LIN {X 0,Y 370.428,Z 641.717,A -85,B 0,C 180,E1 -12894.345,E2 -12894.345} C_VEL
LIN {X 0,Y 371.468,Z 578.131,A -85,B 0,C 180,E1 -12895.586,E2 -12895.586} C_VEL
LIN {X 0,Y 367.34,Z 559.666,A -85,B 0,C 180,E1 -12896.25,E2 -12896.25} C_VEL
LIN {X 0,Y 364.561,Z 552.172,A -85,B 0,C 180,E1 -12896.629,E2 -12896.629} C_VEL
LIN {X 0,Y 362.723,Z 543.261,A -85,B 0,C 180,E1 -12899.318,E2 -12899.318} C_VEL
LIN {X 0,Y 361.889,Z 539.398,A -85,B 0,C 180,E1 -12900.555,E2 -12900.555} C_VEL
LIN {X 0,Y 361.854,Z 539.415,A -85,B 0,C 180,E1 -12904.279,E2 -12904.279} C_VEL
LIN {X 0,Y 361.865,Z 539.408,A -85,B 0,C 180,E1 -12907.222,E2 -12907.222} C_VEL
LIN {X 0,Y 361.904,Z 539.408,A -85,B 0,C 180,E1 -12910.767,E2 -12910.767} C_VEL
LIN {X 0,Y 361.909,Z 539.405,A -85,B 0,C 180,E1 -12914.353,E2 -12914.353} C_VEL
LIN {X 0,Y 361.854,Z 539.407,A -85,B 0,C 180,E1 -12917.563,E2 -12917.563} C_VEL
LIN {X 0,Y 361.87,Z 539.41,A -85,B 0,C 180,E1 -12920.972,E2 -12920.972} C_VEL
LIN {X 0,Y 361.87,Z 539.412,A -85,B 0,C 180,E1 -12924.654,E2 -12924.654} C_VEL
LIN {X 0,Y 361.833,Z 539.415,A -85,B 0,C 180,E1 -12928.37,E2 -12928.37} C_VEL
LIN {X 0,Y 361.897,Z 539.407,A -85,B 0,C 180,E1 -12930.955,E2 -12930.955} C_VEL
LIN {X 0,Y 361.949,Z 539.391,A -85,B 0,C 180,E1 -12933.474,E2 -12933.474} C_VEL
LIN {X 0,Y 361.883,Z 539.4,A -85,B 0,C 180,E1 -12937.144,E2 -12937.144} C_VEL
LIN {X 0,Y 361.899,Z 539.405,A -85,B 0,C 180,E1 -12940.723,E2 -12940.723} C_VEL
LIN {X 0,Y 361.925,Z 539.4,A -85,B 0,C 180,E1 -12943.065,E2 -12943.065} C_VEL
LIN {X 0,Y 361.991,Z 539.389,A -85,B 0,C 180,E1 -12946.527,E2 -12946.527} C_VEL
LIN {X 0,Y 362.024,Z 539.388,A -85,B 0,C 180,E1 -12949.938,E2 -12949.938} C_VEL
LIN {X 0,Y 362.155,Z 539.368,A -85,B 0,C 180,E1 -12953.313,E2 -12953.313} C_VEL
LIN {X 0,Y 362.275,Z 539.348,A -85,B 0,C 180,E1 -12957.776,E2 -12957.776} C_VEL
LIN {X 0,Y 362.421,Z 539.338,A -85,B 0,C 180,E1 -12960,E2 -12960} C_VEL
LIN {X 0,Y 362.274,Z 539.357,A -85,B 0,C 180,E1 -12962.223,E2 -12962.223} C_VEL
LIN {X 0,Y 362.154,Z 539.373,A -85,B 0,C 180,E1 -12966.686,E2 -12966.686} C_VEL
LIN {X 0,Y 362.023,Z 539.385,A -85,B 0,C 180,E1 -12970.062,E2 -12970.062} C_VEL
LIN {X 0,Y 361.99,Z 539.384,A -85,B 0,C 180,E1 -12973.899,E2 -12973.899} C_VEL
LIN {X 0,Y 361.96,Z 539.393,A -85,B 0,C 180,E1 -12977.939,E2 -12977.939} C_VEL
LIN {X 0,Y 361.854,Z 539.408,A -85,B 0,C 180,E1 -12981.655,E2 -12981.655} C_VEL
LIN {X 0,Y 361.92,Z 539.4,A -85,B 0,C 180,E1 -12985.291,E2 -12985.291} C_VEL
LIN {X 0,Y 361.916,Z 539.395,A -85,B 0,C 180,E1 -12987.778,E2 -12987.778} C_VEL
LIN {X 0,Y 361.841,Z 539.41,A -85,B 0,C 180,E1 -12991.286,E2 -12991.286} C_VEL
LIN {X 0,Y 361.849,Z 539.412,A -85,B 0,C 180,E1 -12994.281,E2 -12994.281} C_VEL
LIN {X 0,Y 361.86,Z 539.408,A -85,B 0,C 180,E1 -12997.224,E2 -12997.224} C_VEL
LIN {X 0,Y 361.868,Z 539.411,A -85,B 0,C 180,E1 -13000.763,E2 -13000.763} C_VEL
LIN {X 0,Y 361.861,Z 539.412,A -85,B 0,C 180,E1 -13004.362,E2 -13004.362} C_VEL
LIN {X 0,Y 361.833,Z 539.413,A -85,B 0,C 180,E1 -13007.569,E2 -13007.569} C_VEL
LIN {X 0,Y 361.868,Z 539.411,A -85,B 0,C 180,E1 -13010.974,E2 -13010.974} C_VEL
LIN {X 0,Y 361.872,Z 539.408,A -85,B 0,C 180,E1 -13014.656,E2 -13014.656} C_VEL
LIN {X 0,Y 361.836,Z 539.416,A -85,B 0,C 180,E1 -13018.371,E2 -13018.371} C_VEL
LIN {X 0,Y 361.912,Z 539.551,A -85,B 0,C 180,E1 -13019.371,E2 -13019.371} C_VEL
LIN {X 0,Y 364.641,Z 551.604,A -85,B 0,C 180,E1 -13022.698,E2 -13022.698} C_VEL
LIN {X 0,Y 366.223,Z 560.485,A -85,B 0,C 180,E1 -13025.028,E2 -13025.028} C_VEL
LIN {X 0,Y 365.183,Z 571.057,A -85,B 0,C 180,E1 -13027.484,E2 -13027.484} C_VEL
LIN {X 0,Y 370.275,Z 598.191,A -85,B 0,C 180,E1 -13028.394,E2 -13028.394} C_VEL
LIN {X 0,Y 371.148,Z 604.978,A -85,B 0,C 180,E1 -13028.591,E2 -13028.591} C_VEL
LIN {X 0,Y 369.787,Z 679.549,A -85,B 0,C 180,E1 -13030.068,E2 -13030.068} C_VEL
LIN {X 0,Y 369.085,Z 693.347,A -85,B 0,C 180,E1 -13030.572,E2 -13030.572} C_VEL
LIN {X 0,Y 368.192,Z 705.186,A -85,B 0,C 180,E1 -13031.21,E2 -13031.21} C_VEL
LIN {X 0,Y 367.163,Z 716.398,A -85,B 0,C 180,E1 -13032.022,E2 -13032.022} C_VEL
LIN {X 0,Y 365.9,Z 728.011,A -85,B 0,C 180,E1 -13033.112,E2 -13033.112} C_VEL
LIN {X 0,Y 364.719,Z 738.465,A -85,B 0,C 180,E1 -13034.35,E2 -13034.35} C_VEL
LIN {X 0,Y 363.708,Z 747.897,A -85,B 0,C 180,E1 -13035.738,E2 -13035.738} C_VEL
LIN {X 0,Y 362.56,Z 756.994,A -85,B 0,C 180,E1 -13037.404,E2 -13037.404} C_VEL
LIN {X 0,Y 361.706,Z 764.336,A -85,B 0,C 180,E1 -13039.08,E2 -13039.08} C_VEL
LIN {X 0,Y 361.013,Z 771.091,A -85,B 0,C 180,E1 -13041.041,E2 -13041.041} C_VEL
LIN {X 0,Y 360.601,Z 775.559,A -85,B 0,C 180,E1 -13042.722,E2 -13042.722} C_VEL
LIN {X 0,Y 360.383,Z 778.956,A -85,B 0,C 180,E1 -13044.404,E2 -13044.404} C_VEL
LIN {X 0,Y 360.368,Z 780.651,A -85,B 0,C 180,E1 -13045.526,E2 -13045.526} C_VEL
LIN {X 0,Y 360.3,Z 781.942,A -85,B 0,C 180,E1 -13046.645,E2 -13046.645} C_VEL
LIN {X 0,Y 360.263,Z 782.842,A -85,B 0,C 180,E1 -13047.764,E2 -13047.764} C_VEL
LIN {X 0,Y 360.316,Z 783.319,A -85,B 0,C 180,E1 -13048.882,E2 -13048.882} C_VEL
LIN {X 0,Y 360.359,Z 783.388,A -85,B 0,C 180,E1 -13050,E2 -13050} C_VEL
LIN {X 0,Y 360.317,Z 783.068,A -85,B 0,C 180,E1 -13051.118,E2 -13051.118} C_VEL
LIN {X 0,Y 360.267,Z 782.362,A -85,B 0,C 180,E1 -13052.236,E2 -13052.236} C_VEL
LIN {X 0,Y 360.302,Z 781.236,A -85,B 0,C 180,E1 -13053.355,E2 -13053.355} C_VEL
LIN {X 0,Y 360.368,Z 779.672,A -85,B 0,C 180,E1 -13054.474,E2 -13054.474} C_VEL
LIN {X 0,Y 360.38,Z 776.953,A -85,B 0,C 180,E1 -13055.964,E2 -13055.964} C_VEL
LIN {X 0,Y 360.672,Z 772.311,A -85,B 0,C 180,E1 -13057.839,E2 -13057.839} C_VEL
LIN {X 0,Y 361.163,Z 765.895,A -85,B 0,C 180,E1 -13059.803,E2 -13059.803} C_VEL
LIN {X 0,Y 361.776,Z 758.895,A -85,B 0,C 180,E1 -13061.485,E2 -13061.485} C_VEL
LIN {X 0,Y 362.736,Z 750.12,A -85,B 0,C 180,E1 -13063.159,E2 -13063.159} C_VEL
LIN {X 0,Y 363.645,Z 741.125,A -85,B 0,C 180,E1 -13064.551,E2 -13064.551} C_VEL
LIN {X 0,Y 364.512,Z 731.227,A -85,B 0,C 180,E1 -13065.803,E2 -13065.803} C_VEL
LIN {X 0,Y 365.496,Z 720.293,A -85,B 0,C 180,E1 -13066.907,E2 -13066.907} C_VEL
LIN {X 0,Y 366.567,Z 708.023,A -85,B 0,C 180,E1 -13067.864,E2 -13067.864} C_VEL
LIN {X 0,Y 367.327,Z 696.44,A -85,B 0,C 180,E1 -13068.547,E2 -13068.547} C_VEL
LIN {X 0,Y 367.994,Z 684.292,A -85,B 0,C 180,E1 -13069.053,E2 -13069.053} C_VEL
LIN {X 0,Y 368.341,Z 670.698,A -85,B 0,C 180,E1 -13069.397,E2 -13069.397} C_VEL
LIN {X 0,Y 369.31,Z 603.202,A -85,B 0,C 180,E1 -13070.703,E2 -13070.703} C_VEL
LIN {X 0,Y 364.289,Z 570.9,A -85,B 0,C 180,E1 -13071.65,E2 -13071.65} C_VEL
LIN {X 0,Y 365.458,Z 558.977,A -85,B 0,C 180,E1 -13074.422,E2 -13074.422} C_VEL
LIN {X 0,Y 364.826,Z 553.825,A -85,B 0,C 180,E1 -13075.697,E2 -13075.697} C_VEL
LIN {X 0,Y 362.245,Z 541.043,A -85,B 0,C 180,E1 -13079.014,E2 -13079.014} C_VEL
LIN {X 0,Y 361.912,Z 539.406,A -85,B 0,C 180,E1 -13079.505,E2 -13079.505} C_VEL
LIN {X 0,Y 361.857,Z 539.412,A -85,B 0,C 180,E1 -13083.369,E2 -13083.369} C_VEL
LIN {X 0,Y 361.87,Z 539.407,A -85,B 0,C 180,E1 -13087.017,E2 -13087.017} C_VEL
LIN {X 0,Y 361.853,Z 539.41,A -85,B 0,C 180,E1 -13089.86,E2 -13089.86} C_VEL
LIN {X 0,Y 361.833,Z 539.411,A -85,B 0,C 180,E1 -13092.828,E2 -13092.828} C_VEL
LIN {X 0,Y 361.853,Z 539.409,A -85,B 0,C 180,E1 -13095.939,E2 -13095.939} C_VEL
LIN {X 0,Y 361.868,Z 539.409,A -85,B 0,C 180,E1 -13099.237,E2 -13099.237} C_VEL
LIN {X 0,Y 361.864,Z 539.408,A -85,B 0,C 180,E1 -13102.982,E2 -13102.982} C_VEL
LIN {X 0,Y 361.853,Z 539.407,A -85,B 0,C 180,E1 -13106.63,E2 -13106.63} C_VEL
LIN {X 0,Y 361.87,Z 539.409,A -85,B 0,C 180,E1 -13109.672,E2 -13109.672} C_VEL
LIN {X 0,Y 361.948,Z 539.402,A -85,B 0,C 180,E1 -13113.475,E2 -13113.475} C_VEL
LIN {X 0,Y 361.875,Z 539.408,A -85,B 0,C 180,E1 -13117.144,E2 -13117.144} C_VEL
LIN {X 0,Y 361.913,Z 539.4,A -85,B 0,C 180,E1 -13120.724,E2 -13120.724} C_VEL
LIN {X 0,Y 361.938,Z 539.397,A -85,B 0,C 180,E1 -13124.226,E2 -13124.226} C_VEL
LIN {X 0,Y 361.991,Z 539.39,A -85,B 0,C 180,E1 -13126.528,E2 -13126.528} C_VEL
LIN {X 0,Y 362.023,Z 539.388,A -85,B 0,C 180,E1 -13129.938,E2 -13129.938} C_VEL
LIN {X 0,Y 362.156,Z 539.375,A -85,B 0,C 180,E1 -13133.314,E2 -13133.314} C_VEL
LIN {X 0,Y 362.275,Z 539.358,A -85,B 0,C 180,E1 -13137.777,E2 -13137.777} C_VEL
LIN {X 0,Y 362.419,Z 539.338,A -85,B 0,C 180,E1 -13140,E2 -13140} C_VEL
LIN {X 0,Y 362.275,Z 539.355,A -85,B 0,C 180,E1 -13142.224,E2 -13142.224} C_VEL
LIN {X 0,Y 362.156,Z 539.37,A -85,B 0,C 180,E1 -13146.687,E2 -13146.687} C_VEL
LIN {X 0,Y 362.024,Z 539.387,A -85,B 0,C 180,E1 -13150.062,E2 -13150.062} C_VEL
LIN {X 0,Y 361.99,Z 539.392,A -85,B 0,C 180,E1 -13153.899,E2 -13153.899} C_VEL
LIN {X 0,Y 361.96,Z 539.395,A -85,B 0,C 180,E1 -13157.939,E2 -13157.939} C_VEL
LIN {X 0,Y 361.887,Z 539.407,A -85,B 0,C 180,E1 -13161.654,E2 -13161.654} C_VEL
LIN {X 0,Y 361.922,Z 539.404,A -85,B 0,C 180,E1 -13165.291,E2 -13165.291} C_VEL
LIN {X 0,Y 361.917,Z 539.402,A -85,B 0,C 180,E1 -13167.779,E2 -13167.779} C_VEL
LIN {X 0,Y 361.842,Z 539.414,A -85,B 0,C 180,E1 -13171.286,E2 -13171.286} C_VEL
LIN {X 0,Y 361.85,Z 539.408,A -85,B 0,C 180,E1 -13174.281,E2 -13174.281} C_VEL
LIN {X 0,Y 361.867,Z 539.41,A -85,B 0,C 180,E1 -13177.225,E2 -13177.225} C_VEL
LIN {X 0,Y 361.833,Z 539.411,A -85,B 0,C 180,E1 -13180.757,E2 -13180.757} C_VEL
LIN {X 0,Y 361.844,Z 539.408,A -85,B 0,C 180,E1 -13184.365,E2 -13184.365} C_VEL
LIN {X 0,Y 361.882,Z 539.409,A -85,B 0,C 180,E1 -13187.561,E2 -13187.561} C_VEL
LIN {X 0,Y 361.874,Z 539.407,A -85,B 0,C 180,E1 -13190.973,E2 -13190.973} C_VEL
LIN {X 0,Y 361.874,Z 539.405,A -85,B 0,C 180,E1 -13194.656,E2 -13194.656} C_VEL
LIN {X 0,Y 361.837,Z 539.409,A -85,B 0,C 180,E1 -13198.371,E2 -13198.371} C_VEL
LIN {X 0,Y 361.901,Z 539.403,A -85,B 0,C 180,E1 -13200.956,E2 -13200.956} C_VEL
LIN {X 0,Y 361.956,Z 539.4,A -85,B 0,C 180,E1 -13203.476,E2 -13203.476} C_VEL
LIN {X 0,Y 361.892,Z 539.406,A -85,B 0,C 180,E1 -13207.145,E2 -13207.145} C_VEL
LIN {X 0,Y 361.903,Z 539.507,A -85,B 0,C 180,E1 -13208.772,E2 -13208.772} C_VEL
LIN {X 0,Y 363.757,Z 548.685,A -85,B 0,C 180,E1 -13211.465,E2 -13211.465} C_VEL
LIN {X 0,Y 364.348,Z 552.074,A -85,B 0,C 180,E1 -13212.431,E2 -13212.431} C_VEL
LIN {X 0,Y 366.507,Z 560.951,A -85,B 0,C 180,E1 -13212.742,E2 -13212.742} C_VEL
LIN {X 0,Y 369.698,Z 577.539,A -85,B 0,C 180,E1 -13213.256,E2 -13213.256} C_VEL
LIN {X 0,Y 368.433,Z 659.251,A -85,B 0,C 180,E1 -13214.865,E2 -13214.865} C_VEL
LIN {X 0,Y 367.932,Z 671.574,A -85,B 0,C 180,E1 -13215.304,E2 -13215.304} C_VEL
LIN {X 0,Y 367.179,Z 684.929,A -85,B 0,C 180,E1 -13216.016,E2 -13216.016} C_VEL
LIN {X 0,Y 366.354,Z 696.143,A -85,B 0,C 180,E1 -13216.832,E2 -13216.832} C_VEL
LIN {X 0,Y 365.456,Z 707.705,A -85,B 0,C 180,E1 -13217.929,E2 -13217.929} C_VEL
LIN {X 0,Y 364.341,Z 718.119,A -85,B 0,C 180,E1 -13219.16,E2 -13219.16} C_VEL
LIN {X 0,Y 363.471,Z 726.919,A -85,B 0,C 180,E1 -13220.447,E2 -13220.447} C_VEL
LIN {X 0,Y 362.708,Z 735.175,A -85,B 0,C 180,E1 -13221.925,E2 -13221.925} C_VEL
LIN {X 0,Y 361.952,Z 742.691,A -85,B 0,C 180,E1 -13223.59,E2 -13223.59} C_VEL
LIN {X 0,Y 361.489,Z 747.841,A -85,B 0,C 180,E1 -13224.981,E2 -13224.981} C_VEL
LIN {X 0,Y 360.912,Z 752.837,A -85,B 0,C 180,E1 -13226.651,E2 -13226.651} C_VEL
LIN {X 0,Y 360.63,Z 756.711,A -85,B 0,C 180,E1 -13228.325,E2 -13228.325} C_VEL
LIN {X 0,Y 360.435,Z 759.571,A -85,B 0,C 180,E1 -13230,E2 -13230} C_VEL
LIN {X 0,Y 360.372,Z 760.923,A -85,B 0,C 180,E1 -13231.117,E2 -13231.117} C_VEL
LIN {X 0,Y 360.307,Z 762.469,A -85,B 0,C 180,E1 -13233.355,E2 -13233.355} C_VEL
LIN {X 0,Y 360.337,Z 762.65,A -85,B 0,C 180,E1 -13234.474,E2 -13234.474} C_VEL
LIN {X 0,Y 360.387,Z 761.791,A -85,B 0,C 180,E1 -13236.719,E2 -13236.719} C_VEL
LIN {X 0,Y 360.458,Z 760.786,A -85,B 0,C 180,E1 -13237.844,E2 -13237.844} C_VEL
LIN {X 0,Y 360.563,Z 759.362,A -85,B 0,C 180,E1 -13238.971,E2 -13238.971} C_VEL
LIN {X 0,Y 360.819,Z 756.409,A -85,B 0,C 180,E1 -13240.663,E2 -13240.663} C_VEL
LIN {X 0,Y 361.301,Z 752.402,A -85,B 0,C 180,E1 -13242.355,E2 -13242.355} C_VEL
LIN {X 0,Y 361.886,Z 747.191,A -85,B 0,C 180,E1 -13244.057,E2 -13244.057} C_VEL
LIN {X 0,Y 362.686,Z 740.685,A -85,B 0,C 180,E1 -13245.74,E2 -13245.74} C_VEL
LIN {X 0,Y 363.732,Z 732.542,A -85,B 0,C 180,E1 -13247.427,E2 -13247.427} C_VEL
LIN {X 0,Y 364.811,Z 724.201,A -85,B 0,C 180,E1 -13248.825,E2 -13248.825} C_VEL
LIN {X 0,Y 365.93,Z 713.912,A -85,B 0,C 180,E1 -13250.224,E2 -13250.224} C_VEL
LIN {X 0,Y 367.195,Z 702.254,A -85,B 0,C 180,E1 -13251.471,E2 -13251.471} C_VEL
LIN {X 0,Y 368.295,Z 690.699,A -85,B 0,C 180,E1 -13252.435,E2 -13252.435} C_VEL
LIN {X 0,Y 369.137,Z 678.654,A -85,B 0,C 180,E1 -13253.195,E2 -13253.195} C_VEL
LIN {X 0,Y 369.331,Z 674.63,A -85,B 0,C 180,E1 -13253.406,E2 -13253.406} C_VEL
LIN {X 0,Y 369.243,Z 668.987,A -85,B 0,C 180,E1 -13253.678,E2 -13253.678} C_VEL
LIN {X 0,Y 367.049,Z 659.817,A -85,B 0,C 180,E1 -13254.149,E2 -13254.149} C_VEL
LIN {X 0,Y 364.45,Z 650.556,A -85,B 0,C 180,E1 -13254.544,E2 -13254.544} C_VEL
LIN {X 0,Y 363.836,Z 644.759,A -85,B 0,C 180,E1 -13254.703,E2 -13254.703} C_VEL
LIN {X 0,Y 364.96,Z 579.185,A -85,B 0,C 180,E1 -13256.005,E2 -13256.005} C_VEL
LIN {X 0,Y 361.216,Z 562.272,A -85,B 0,C 180,E1 -13256.628,E2 -13256.628} C_VEL
LIN {X 0,Y 357.409,Z 552.439,A -85,B 0,C 180,E1 -13257.132,E2 -13257.132} C_VEL
LIN {X 0,Y 355.718,Z 544.387,A -85,B 0,C 180,E1 -13259.62,E2 -13259.62} C_VEL
LIN {X 0,Y 354.829,Z 540.277,A -85,B 0,C 180,E1 -13260.995,E2 -13260.995} C_VEL
LIN {X 0,Y 354.812,Z 540.287,A -85,B 0,C 180,E1 -13265.058,E2 -13265.058} C_VEL
LIN {X 0,Y 354.807,Z 540.285,A -85,B 0,C 180,E1 -13267.882,E2 -13267.882} C_VEL
LIN {X 0,Y 354.837,Z 540.284,A -85,B 0,C 180,E1 -13271.18,E2 -13271.18} C_VEL
LIN {X 0,Y 354.861,Z 540.284,A -85,B 0,C 180,E1 -13274.522,E2 -13274.522} C_VEL
LIN {X 0,Y 354.811,Z 540.284,A -85,B 0,C 180,E1 -13277.665,E2 -13277.665} C_VEL
LIN {X 0,Y 354.834,Z 540.283,A -85,B 0,C 180,E1 -13280.668,E2 -13280.668} C_VEL
LIN {X 0,Y 354.818,Z 540.287,A -85,B 0,C 180,E1 -13284.3,E2 -13284.3} C_VEL
LIN {X 0,Y 354.782,Z 540.29,A -85,B 0,C 180,E1 -13287.666,E2 -13287.666} C_VEL
LIN {X 0,Y 354.864,Z 540.28,A -85,B 0,C 180,E1 -13290.62,E2 -13290.62} C_VEL
LIN {X 0,Y 354.893,Z 540.272,A -85,B 0,C 180,E1 -13294.172,E2 -13294.172} C_VEL
LIN {X 0,Y 354.828,Z 540.277,A -85,B 0,C 180,E1 -13297.893,E2 -13297.893} C_VEL
LIN {X 0,Y 354.915,Z 540.269,A -85,B 0,C 180,E1 -13301.891,E2 -13301.891} C_VEL
LIN {X 0,Y 354.935,Z 540.27,A -85,B 0,C 180,E1 -13305.981,E2 -13305.981} C_VEL
LIN {X 0,Y 354.97,Z 540.266,A -85,B 0,C 180,E1 -13309.735,E2 -13309.735} C_VEL
LIN {X 0,Y 355.118,Z 540.246,A -85,B 0,C 180,E1 -13313.18,E2 -13313.18} C_VEL
LIN {X 0,Y 355.238,Z 540.224,A -85,B 0,C 180,E1 -13317.732,E2 -13317.732} C_VEL
LIN {X 0,Y 355.391,Z 540.213,A -85,B 0,C 180,E1 -13320,E2 -13320} C_VEL
LIN {X 0,Y 355.238,Z 540.232,A -85,B 0,C 180,E1 -13322.268,E2 -13322.268} C_VEL
LIN {X 0,Y 355.118,Z 540.248,A -85,B 0,C 180,E1 -13326.819,E2 -13326.819} C_VEL
LIN {X 0,Y 354.97,Z 540.266,A -85,B 0,C 180,E1 -13330.264,E2 -13330.264} C_VEL
LIN {X 0,Y 354.935,Z 540.263,A -85,B 0,C 180,E1 -13334.019,E2 -13334.019} C_VEL
LIN {X 0,Y 354.916,Z 540.271,A -85,B 0,C 180,E1 -13338.109,E2 -13338.109} C_VEL
LIN {X 0,Y 354.809,Z 540.287,A -85,B 0,C 180,E1 -13342.108,E2 -13342.108} C_VEL
LIN {X 0,Y 354.892,Z 540.276,A -85,B 0,C 180,E1 -13345.828,E2 -13345.828} C_VEL
LIN {X 0,Y 354.848,Z 540.281,A -85,B 0,C 180,E1 -13349.679,E2 -13349.679} C_VEL
LIN {X 0,Y 354.801,Z 540.287,A -85,B 0,C 180,E1 -13353.703,E2 -13353.703} C_VEL
LIN {X 0,Y 354.794,Z 540.292,A -85,B 0,C 180,E1 -13356.46,E2 -13356.46} C_VEL
LIN {X 0,Y 354.819,Z 540.285,A -85,B 0,C 180,E1 -13359.424,E2 -13359.424} C_VEL
LIN {X 0,Y 354.801,Z 540.292,A -85,B 0,C 180,E1 -13362.871,E2 -13362.871} C_VEL
LIN {X 0,Y 354.766,Z 540.294,A -85,B 0,C 180,E1 -13366.105,E2 -13366.105} C_VEL
LIN {X 0,Y 354.786,Z 540.291,A -85,B 0,C 180,E1 -13369.18,E2 -13369.18} C_VEL
LIN {X 0,Y 354.806,Z 540.287,A -85,B 0,C 180,E1 -13372.403,E2 -13372.403} C_VEL
LIN {X 0,Y 354.81,Z 540.289,A -85,B 0,C 180,E1 -13374.942,E2 -13374.942} C_VEL
LIN {X 0,Y 354.832,Z 540.386,A -85,B 0,C 180,E1 -13378.923,E2 -13378.923} C_VEL
LIN {X 0,Y 357.509,Z 551.94,A -85,B 0,C 180,E1 -13382.205,E2 -13382.205} C_VEL
LIN {X 0,Y 359.308,Z 561.667,A -85,B 0,C 180,E1 -13384.823,E2 -13384.823} C_VEL
LIN {X 0,Y 358.399,Z 570.588,A -85,B 0,C 180,E1 -13386.987,E2 -13386.987} C_VEL
LIN {X 0,Y 363.845,Z 599.803,A -85,B 0,C 180,E1 -13387.997,E2 -13387.997} C_VEL
LIN {X 0,Y 364.603,Z 606.653,A -85,B 0,C 180,E1 -13388.193,E2 -13388.193} C_VEL
LIN {X 0,Y 363.197,Z 679.224,A -85,B 0,C 180,E1 -13389.654,E2 -13389.654} C_VEL
LIN {X 0,Y 362.483,Z 693.061,A -85,B 0,C 180,E1 -13390.166,E2 -13390.166} C_VEL
LIN {X 0,Y 361.485,Z 705.467,A -85,B 0,C 180,E1 -13390.848,E2 -13390.848} C_VEL
LIN {X 0,Y 360.263,Z 718.124,A -85,B 0,C 180,E1 -13391.813,E2 -13391.813} C_VEL
LIN {X 0,Y 358.959,Z 729.382,A -85,B 0,C 180,E1 -13392.922,E2 -13392.922} C_VEL
LIN {X 0,Y 357.738,Z 739.73,A -85,B 0,C 180,E1 -13394.211,E2 -13394.211} C_VEL
LIN {X 0,Y 356.614,Z 749.505,A -85,B 0,C 180,E1 -13395.739,E2 -13395.739} C_VEL
LIN {X 0,Y 355.429,Z 758.294,A -85,B 0,C 180,E1 -13397.438,E2 -13397.438} C_VEL
LIN {X 0,Y 354.59,Z 765.335,A -85,B 0,C 180,E1 -13399.147,E2 -13399.147} C_VEL
LIN {X 0,Y 353.96,Z 770.973,A -85,B 0,C 180,E1 -13400.86,E2 -13400.86} C_VEL
LIN {X 0,Y 353.525,Z 775.421,A -85,B 0,C 180,E1 -13402.576,E2 -13402.576} C_VEL
LIN {X 0,Y 353.281,Z 778.799,A -85,B 0,C 180,E1 -13404.292,E2 -13404.292} C_VEL
LIN {X 0,Y 353.28,Z 780.485,A -85,B 0,C 180,E1 -13405.436,E2 -13405.436} C_VEL
LIN {X 0,Y 353.222,Z 781.768,A -85,B 0,C 180,E1 -13406.578,E2 -13406.578} C_VEL
LIN {X 0,Y 353.172,Z 782.658,A -85,B 0,C 180,E1 -13407.719,E2 -13407.719} C_VEL
LIN {X 0,Y 353.216,Z 783.119,A -85,B 0,C 180,E1 -13408.86,E2 -13408.86} C_VEL
LIN {X 0,Y 353.262,Z 783.179,A -85,B 0,C 180,E1 -13410,E2 -13410} C_VEL
LIN {X 0,Y 353.217,Z 782.85,A -85,B 0,C 180,E1 -13411.14,E2 -13411.14} C_VEL
LIN {X 0,Y 353.175,Z 782.135,A -85,B 0,C 180,E1 -13412.281,E2 -13412.281} C_VEL
LIN {X 0,Y 353.224,Z 780.992,A -85,B 0,C 180,E1 -13413.422,E2 -13413.422} C_VEL
LIN {X 0,Y 353.281,Z 779.419,A -85,B 0,C 180,E1 -13414.564,E2 -13414.564} C_VEL
LIN {X 0,Y 353.334,Z 776.252,A -85,B 0,C 180,E1 -13416.28,E2 -13416.28} C_VEL
LIN {X 0,Y 353.616,Z 772.017,A -85,B 0,C 180,E1 -13417.997,E2 -13417.997} C_VEL
LIN {X 0,Y 354.126,Z 765.579,A -85,B 0,C 180,E1 -13420,E2 -13420} C_VEL
LIN {X 0,Y 354.762,Z 758.544,A -85,B 0,C 180,E1 -13421.716,E2 -13421.716} C_VEL
LIN {X 0,Y 355.79,Z 749.734,A -85,B 0,C 180,E1 -13423.42,E2 -13423.42} C_VEL
LIN {X 0,Y 356.75,Z 740.704,A -85,B 0,C 180,E1 -13424.838,E2 -13424.838} C_VEL
LIN {X 0,Y 357.64,Z 730.759,A -85,B 0,C 180,E1 -13426.115,E2 -13426.115} C_VEL
LIN {X 0,Y 358.674,Z 719.735,A -85,B 0,C 180,E1 -13427.239,E2 -13427.239} C_VEL
LIN {X 0,Y 359.781,Z 707.374,A -85,B 0,C 180,E1 -13428.212,E2 -13428.212} C_VEL
LIN {X 0,Y 360.577,Z 695.654,A -85,B 0,C 180,E1 -13428.907,E2 -13428.907} C_VEL
LIN {X 0,Y 361.249,Z 683.125,A -85,B 0,C 180,E1 -13429.423,E2 -13429.423} C_VEL
LIN {X 0,Y 361.716,Z 667.113,A -85,B 0,C 180,E1 -13429.803,E2 -13429.803} C_VEL
LIN {X 0,Y 362.559,Z 603.763,A -85,B 0,C 180,E1 -13431.058,E2 -13431.058} C_VEL
LIN {X 0,Y 357.407,Z 570.783,A -85,B 0,C 180,E1 -13432.037,E2 -13432.037} C_VEL
LIN {X 0,Y 358.505,Z 559.891,A -85,B 0,C 180,E1 -13434.618,E2 -13434.618} C_VEL
LIN {X 0,Y 357.575,Z 553.506,A -85,B 0,C 180,E1 -13436.245,E2 -13436.245} C_VEL
LIN {X 0,Y 355.11,Z 541.491,A -85,B 0,C 180,E1 -13439.447,E2 -13439.447} C_VEL
LIN {X 0,Y 354.845,Z 540.286,A -85,B 0,C 180,E1 -13439.842,E2 -13439.842} C_VEL
LIN {X 0,Y 354.804,Z 540.29,A -85,B 0,C 180,E1 -13443.701,E2 -13443.701} C_VEL
LIN {X 0,Y 354.799,Z 540.286,A -85,B 0,C 180,E1 -13446.458,E2 -13446.458} C_VEL
LIN {X 0,Y 354.821,Z 540.289,A -85,B 0,C 180,E1 -13449.423,E2 -13449.423} C_VEL
LIN {X 0,Y 354.785,Z 540.289,A -85,B 0,C 180,E1 -13452.867,E2 -13452.867} C_VEL
LIN {X 0,Y 354.798,Z 540.287,A -85,B 0,C 180,E1 -13456.108,E2 -13456.108} C_VEL
LIN {X 0,Y 354.82,Z 540.287,A -85,B 0,C 180,E1 -13459.183,E2 -13459.183} C_VEL
LIN {X 0,Y 354.804,Z 540.285,A -85,B 0,C 180,E1 -13462.401,E2 -13462.401} C_VEL
LIN {X 0,Y 354.807,Z 540.287,A -85,B 0,C 180,E1 -13464.94,E2 -13464.94} C_VEL
LIN {X 0,Y 354.787,Z 540.287,A -85,B 0,C 180,E1 -13468.405,E2 -13468.405} C_VEL
LIN {X 0,Y 354.847,Z 540.285,A -85,B 0,C 180,E1 -13471.619,E2 -13471.619} C_VEL
LIN {X 0,Y 354.892,Z 540.275,A -85,B 0,C 180,E1 -13474.172,E2 -13474.172} C_VEL
LIN {X 0,Y 354.81,Z 540.287,A -85,B 0,C 180,E1 -13477.892,E2 -13477.892} C_VEL
LIN {X 0,Y 354.916,Z 540.273,A -85,B 0,C 180,E1 -13481.891,E2 -13481.891} C_VEL
LIN {X 0,Y 354.935,Z 540.271,A -85,B 0,C 180,E1 -13485.981,E2 -13485.981} C_VEL
LIN {X 0,Y 354.97,Z 540.268,A -85,B 0,C 180,E1 -13489.736,E2 -13489.736} C_VEL
LIN {X 0,Y 355.12,Z 540.25,A -85,B 0,C 180,E1 -13493.181,E2 -13493.181} C_VEL
LIN {X 0,Y 355.238,Z 540.235,A -85,B 0,C 180,E1 -13497.732,E2 -13497.732} C_VEL
LIN {X 0,Y 355.389,Z 540.214,A -85,B 0,C 180,E1 -13500,E2 -13500} C_VEL
LIN {X 0,Y 355.238,Z 540.231,A -85,B 0,C 180,E1 -13502.268,E2 -13502.268} C_VEL
LIN {X 0,Y 355.119,Z 540.247,A -85,B 0,C 180,E1 -13506.82,E2 -13506.82} C_VEL
LIN {X 0,Y 354.97,Z 540.264,A -85,B 0,C 180,E1 -13510.265,E2 -13510.265} C_VEL
LIN {X 0,Y 354.935,Z 540.27,A -85,B 0,C 180,E1 -13514.019,E2 -13514.019} C_VEL
LIN {X 0,Y 354.915,Z 540.272,A -85,B 0,C 180,E1 -13518.109,E2 -13518.109} C_VEL
LIN {X 0,Y 354.829,Z 540.283,A -85,B 0,C 180,E1 -13522.107,E2 -13522.107} C_VEL
LIN {X 0,Y 354.893,Z 540.276,A -85,B 0,C 180,E1 -13525.828,E2 -13525.828} C_VEL
LIN {X 0,Y 354.849,Z 540.283,A -85,B 0,C 180,E1 -13529.679,E2 -13529.679} C_VEL
LIN {X 0,Y 354.802,Z 540.289,A -85,B 0,C 180,E1 -13533.703,E2 -13533.703} C_VEL
LIN {X 0,Y 354.797,Z 540.286,A -85,B 0,C 180,E1 -13536.46,E2 -13536.46} C_VEL
LIN {X 0,Y 354.82,Z 540.29,A -85,B 0,C 180,E1 -13539.425,E2 -13539.425} C_VEL
LIN {X 0,Y 354.788,Z 540.289,A -85,B 0,C 180,E1 -13542.869,E2 -13542.869} C_VEL
LIN {X 0,Y 354.849,Z 540.28,A -85,B 0,C 180,E1 -13546.118,E2 -13546.118} C_VEL
LIN {X 0,Y 354.855,Z 540.283,A -85,B 0,C 180,E1 -13549.19,E2 -13549.19} C_VEL
LIN {X 0,Y 354.808,Z 540.285,A -85,B 0,C 180,E1 -13552.403,E2 -13552.403} C_VEL
LIN {X 0,Y 354.812,Z 540.286,A -85,B 0,C 180,E1 -13554.942,E2 -13554.942} C_VEL
LIN {X 0,Y 354.793,Z 540.287,A -85,B 0,C 180,E1 -13558.406,E2 -13558.406} C_VEL
LIN {X 0,Y 354.852,Z 540.284,A -85,B 0,C 180,E1 -13561.62,E2 -13561.62} C_VEL
LIN {X 0,Y 354.901,Z 540.274,A -85,B 0,C 180,E1 -13564.173,E2 -13564.173} C_VEL
LIN {X 0,Y 354.879,Z 540.369,A -85,B 0,C 180,E1 -13568.471,E2 -13568.471} C_VEL
LIN {X 0,Y 356.64,Z 549.028,A -85,B 0,C 180,E1 -13571.067,E2 -13571.067} C_VEL
LIN {X 0,Y 357.231,Z 552.349,A -85,B 0,C 180,E1 -13572.021,E2 -13572.021} C_VEL
LIN {X 0,Y 359.465,Z 560.119,A -85,B 0,C 180,E1 -13572.318,E2 -13572.318} C_VEL
LIN {X 0,Y 363.012,Z 578.792,A -85,B 0,C 180,E1 -13572.91,E2 -13572.91} C_VEL
LIN {X 0,Y 361.678,Z 659.895,A -85,B 0,C 180,E1 -13574.54,E2 -13574.54} C_VEL
LIN {X 0,Y 361.157,Z 672.073,A -85,B 0,C 180,E1 -13574.986,E2 -13574.986} C_VEL
LIN {X 0,Y 360.423,Z 684.79,A -85,B 0,C 180,E1 -13575.677,E2 -13575.677} C_VEL
LIN {X 0,Y 359.497,Z 696.895,A -85,B 0,C 180,E1 -13576.577,E2 -13576.577} C_VEL
LIN {X 0,Y 358.557,Z 708.355,A -85,B 0,C 180,E1 -13577.693,E2 -13577.693} C_VEL
LIN {X 0,Y 357.413,Z 718.692,A -85,B 0,C 180,E1 -13578.947,E2 -13578.947} C_VEL
LIN {X 0,Y 356.448,Z 727.966,A -85,B 0,C 180,E1 -13580.348,E2 -13580.348} C_VEL
LIN {X 0,Y 355.568,Z 736.959,A -85,B 0,C 180,E1 -13582.047,E2 -13582.047} C_VEL
LIN {X 0,Y 354.908,Z 743.09,A -85,B 0,C 180,E1 -13583.462,E2 -13583.462} C_VEL
LIN {X 0,Y 354.439,Z 748.202,A -85,B 0,C 180,E1 -13584.881,E2 -13584.881} C_VEL
LIN {X 0,Y 353.833,Z 753.166,A -85,B 0,C 180,E1 -13586.584,E2 -13586.584} C_VEL
LIN {X 0,Y 353.561,Z 757.007,A -85,B 0,C 180,E1 -13588.291,E2 -13588.291} C_VEL
LIN {X 0,Y 353.339,Z 759.839,A -85,B 0,C 180,E1 -13590,E2 -13590} C_VEL
LIN {X 0,Y 353.272,Z 761.177,A -85,B 0,C 180,E1 -13591.14,E2 -13591.14} C_VEL
LIN {X 0,Y 353.227,Z 762.695,A -85,B 0,C 180,E1 -13593.422,E2 -13593.422} C_VEL
LIN {X 0,Y 353.25,Z 762.848,A -85,B 0,C 180,E1 -13594.564,E2 -13594.564} C_VEL
LIN {X 0,Y 353.279,Z 762.513,A -85,B 0,C 180,E1 -13595.908,E2 -13595.908} C_VEL
LIN {X 0,Y 353.398,Z 760.942,A -85,B 0,C 180,E1 -13598.002,E2 -13598.002} C_VEL
LIN {X 0,Y 353.505,Z 759.489,A -85,B 0,C 180,E1 -13599.151,E2 -13599.151} C_VEL
LIN {X 0,Y 353.803,Z 756.508,A -85,B 0,C 180,E1 -13600.877,E2 -13600.877} C_VEL
LIN {X 0,Y 354.281,Z 752.469,A -85,B 0,C 180,E1 -13602.604,E2 -13602.604} C_VEL
LIN {X 0,Y 355.029,Z 746.341,A -85,B 0,C 180,E1 -13604.59,E2 -13604.59} C_VEL
LIN {X 0,Y 355.951,Z 739.442,A -85,B 0,C 180,E1 -13606.341,E2 -13606.341} C_VEL
LIN {X 0,Y 357.133,Z 730.942,A -85,B 0,C 180,E1 -13608.055,E2 -13608.055} C_VEL
LIN {X 0,Y 358.222,Z 722.171,A -85,B 0,C 180,E1 -13609.482,E2 -13609.482} C_VEL
LIN {X 0,Y 359.501,Z 711.348,A -85,B 0,C 180,E1 -13610.902,E2 -13610.902} C_VEL
LIN {X 0,Y 360.697,Z 700.464,A -85,B 0,C 180,E1 -13612.028,E2 -13612.028} C_VEL
LIN {X 0,Y 361.793,Z 689.219,A -85,B 0,C 180,E1 -13612.937,E2 -13612.937} C_VEL
LIN {X 0,Y 362.586,Z 676.635,A -85,B 0,C 180,E1 -13613.715,E2 -13613.715} C_VEL
LIN {X 0,Y 363.31,Z 664.117,A -85,B 0,C 180,E1 -13614.246,E2 -13614.246} C_VEL
LIN {X 0,Y 363.755,Z 648.877,A -85,B 0,C 180,E1 -13614.623,E2 -13614.623} C_VEL
LIN {X 0,Y 363.836,Z 644.759,A -85,B 0,C 180,E1 -13614.703,E2 -13614.703} C_VEL
LIN {X 0,Y 363.289,Z 638.956,A -85,B 0,C 180,E1 -13614.861,E2 -13614.861} C_VEL
LIN {X 0,Y 358.356,Z 620.289,A -85,B 0,C 180,E1 -13615.589,E2 -13615.589} C_VEL
LIN {X 0,Y 357.836,Z 614.486,A -85,B 0,C 180,E1 -13615.749,E2 -13615.749} C_VEL
LIN {X 0,Y 358.484,Z 580.193,A -85,B 0,C 180,E1 -13616.44,E2 -13616.44} C_VEL
LIN {X 0,Y 354.892,Z 564.372,A -85,B 0,C 180,E1 -13617.046,E2 -13617.046} C_VEL
LIN {X 0,Y 350.281,Z 552.671,A -85,B 0,C 180,E1 -13617.664,E2 -13617.664} C_VEL
LIN {X 0,Y 347.772,Z 541.158,A -85,B 0,C 180,E1 -13621.356,E2 -13621.356} C_VEL
LIN {X 0,Y 347.744,Z 541.172,A -85,B 0,C 180,E1 -13624.463,E2 -13624.463} C_VEL
LIN {X 0,Y 347.775,Z 541.161,A -85,B 0,C 180,E1 -13627.988,E2 -13627.988} C_VEL
LIN {X 0,Y 347.782,Z 541.161,A -85,B 0,C 180,E1 -13631.608,E2 -13631.608} C_VEL
LIN {X 0,Y 347.796,Z 541.161,A -85,B 0,C 180,E1 -13635.011,E2 -13635.011} C_VEL
LIN {X 0,Y 347.765,Z 541.156,A -85,B 0,C 180,E1 -13638.393,E2 -13638.393} C_VEL
LIN {X 0,Y 347.775,Z 541.164,A -85,B 0,C 180,E1 -13642.009,E2 -13642.009} C_VEL
LIN {X 0,Y 347.74,Z 541.165,A -85,B 0,C 180,E1 -13645.535,E2 -13645.535} C_VEL
LIN {X 0,Y 347.759,Z 541.159,A -85,B 0,C 180,E1 -13649.653,E2 -13649.653} C_VEL
LIN {X 0,Y 347.847,Z 541.152,A -85,B 0,C 180,E1 -13652.744,E2 -13652.744} C_VEL
LIN {X 0,Y 347.782,Z 541.163,A -85,B 0,C 180,E1 -13656.161,E2 -13656.161} C_VEL
LIN {X 0,Y 347.806,Z 541.159,A -85,B 0,C 180,E1 -13659.909,E2 -13659.909} C_VEL
LIN {X 0,Y 347.859,Z 541.148,A -85,B 0,C 180,E1 -13662.359,E2 -13662.359} C_VEL
LIN {X 0,Y 347.891,Z 541.148,A -85,B 0,C 180,E1 -13665.97,E2 -13665.97} C_VEL
LIN {X 0,Y 347.921,Z 541.144,A -85,B 0,C 180,E1 -13669.525,E2 -13669.525} C_VEL
LIN {X 0,Y 348.084,Z 541.121,A -85,B 0,C 180,E1 -13673.042,E2 -13673.042} C_VEL
LIN {X 0,Y 348.201,Z 541.101,A -85,B 0,C 180,E1 -13677.686,E2 -13677.686} C_VEL
LIN {X 0,Y 348.36,Z 541.089,A -85,B 0,C 180,E1 -13680,E2 -13680} C_VEL
LIN {X 0,Y 348.2,Z 541.108,A -85,B 0,C 180,E1 -13682.313,E2 -13682.313} C_VEL
LIN {X 0,Y 348.084,Z 541.123,A -85,B 0,C 180,E1 -13686.958,E2 -13686.958} C_VEL
LIN {X 0,Y 347.921,Z 541.146,A -85,B 0,C 180,E1 -13690.475,E2 -13690.475} C_VEL
LIN {X 0,Y 347.891,Z 541.141,A -85,B 0,C 180,E1 -13694.15,E2 -13694.15} C_VEL
LIN {X 0,Y 347.884,Z 541.146,A -85,B 0,C 180,E1 -13698.291,E2 -13698.291} C_VEL
LIN {X 0,Y 347.761,Z 541.163,A -85,B 0,C 180,E1 -13701.627,E2 -13701.627} C_VEL
LIN {X 0,Y 347.805,Z 541.16,A -85,B 0,C 180,E1 -13705.109,E2 -13705.109} C_VEL
LIN {X 0,Y 347.806,Z 541.153,A -85,B 0,C 180,E1 -13707.694,E2 -13707.694} C_VEL
LIN {X 0,Y 347.758,Z 541.167,A -85,B 0,C 180,E1 -13710.347,E2 -13710.347} C_VEL
LIN {X 0,Y 347.739,Z 541.17,A -85,B 0,C 180,E1 -13714.465,E2 -13714.465} C_VEL
LIN {X 0,Y 347.771,Z 541.164,A -85,B 0,C 180,E1 -13717.99,E2 -13717.99} C_VEL
LIN {X 0,Y 347.762,Z 541.166,A -85,B 0,C 180,E1 -13721.829,E2 -13721.829} C_VEL
LIN {X 0,Y 347.764,Z 541.167,A -85,B 0,C 180,E1 -13725.017,E2 -13725.017} C_VEL
LIN {X 0,Y 347.748,Z 541.17,A -85,B 0,C 180,E1 -13728.398,E2 -13728.398} C_VEL
LIN {X 0,Y 347.772,Z 541.164,A -85,B 0,C 180,E1 -13732.012,E2 -13732.012} C_VEL
LIN {X 0,Y 347.743,Z 541.169,A -85,B 0,C 180,E1 -13735.537,E2 -13735.537} C_VEL
LIN {X 0,Y 347.776,Z 541.279,A -85,B 0,C 180,E1 -13738.474,E2 -13738.474} C_VEL
LIN {X 0,Y 350.34,Z 552.35,A -85,B 0,C 180,E1 -13741.706,E2 -13741.706} C_VEL
LIN {X 0,Y 352.373,Z 562.85,A -85,B 0,C 180,E1 -13744.608,E2 -13744.608} C_VEL
LIN {X 0,Y 351.675,Z 570.39,A -85,B 0,C 180,E1 -13746.484,E2 -13746.484} C_VEL
LIN {X 0,Y 357.359,Z 600.782,A -85,B 0,C 180,E1 -13747.567,E2 -13747.567} C_VEL
LIN {X 0,Y 358.092,Z 608.172,A -85,B 0,C 180,E1 -13747.778,E2 -13747.778} C_VEL
LIN {X 0,Y 356.647,Z 678.908,A -85,B 0,C 180,E1 -13749.225,E2 -13749.225} C_VEL
LIN {X 0,Y 355.878,Z 692.783,A -85,B 0,C 180,E1 -13749.745,E2 -13749.745} C_VEL
LIN {X 0,Y 354.882,Z 704.662,A -85,B 0,C 180,E1 -13750.402,E2 -13750.402} C_VEL
LIN {X 0,Y 353.734,Z 716.695,A -85,B 0,C 180,E1 -13751.315,E2 -13751.315} C_VEL
LIN {X 0,Y 352.349,Z 728.178,A -85,B 0,C 180,E1 -13752.442,E2 -13752.442} C_VEL
LIN {X 0,Y 351.06,Z 738.532,A -85,B 0,C 180,E1 -13753.724,E2 -13753.724} C_VEL
LIN {X 0,Y 349.888,Z 747.854,A -85,B 0,C 180,E1 -13755.161,E2 -13755.161} C_VEL
LIN {X 0,Y 348.672,Z 756.884,A -85,B 0,C 180,E1 -13756.894,E2 -13756.894} C_VEL
LIN {X 0,Y 347.68,Z 764.172,A -85,B 0,C 180,E1 -13758.634,E2 -13758.634} C_VEL
LIN {X 0,Y 346.922,Z 770.857,A -85,B 0,C 180,E1 -13760.673,E2 -13760.673} C_VEL
LIN {X 0,Y 346.476,Z 775.284,A -85,B 0,C 180,E1 -13762.424,E2 -13762.424} C_VEL
LIN {X 0,Y 346.201,Z 778.643,A -85,B 0,C 180,E1 -13764.174,E2 -13764.174} C_VEL
LIN {X 0,Y 346.175,Z 780.32,A -85,B 0,C 180,E1 -13765.342,E2 -13765.342} C_VEL
LIN {X 0,Y 346.146,Z 781.595,A -85,B 0,C 180,E1 -13766.508,E2 -13766.508} C_VEL
LIN {X 0,Y 346.083,Z 782.473,A -85,B 0,C 180,E1 -13767.672,E2 -13767.672} C_VEL
LIN {X 0,Y 346.116,Z 782.918,A -85,B 0,C 180,E1 -13768.837,E2 -13768.837} C_VEL
LIN {X 0,Y 346.165,Z 782.969,A -85,B 0,C 180,E1 -13770,E2 -13770} C_VEL
LIN {X 0,Y 346.118,Z 782.632,A -85,B 0,C 180,E1 -13771.163,E2 -13771.163} C_VEL
LIN {X 0,Y 346.086,Z 781.908,A -85,B 0,C 180,E1 -13772.328,E2 -13772.328} C_VEL
LIN {X 0,Y 346.148,Z 780.748,A -85,B 0,C 180,E1 -13773.492,E2 -13773.492} C_VEL
LIN {X 0,Y 346.17,Z 777.834,A -85,B 0,C 180,E1 -13775.459,E2 -13775.459} C_VEL
LIN {X 0,Y 346.448,Z 773.272,A -85,B 0,C 180,E1 -13777.577,E2 -13777.577} C_VEL
LIN {X 0,Y 346.818,Z 768.245,A -85,B 0,C 180,E1 -13779.329,E2 -13779.329} C_VEL
LIN {X 0,Y 347.404,Z 761.927,A -85,B 0,C 180,E1 -13781.08,E2 -13781.08} C_VEL
LIN {X 0,Y 348.278,Z 754.008,A -85,B 0,C 180,E1 -13782.825,E2 -13782.825} C_VEL
LIN {X 0,Y 349.179,Z 745.932,A -85,B 0,C 180,E1 -13784.274,E2 -13784.274} C_VEL
LIN {X 0,Y 350.245,Z 735.777,A -85,B 0,C 180,E1 -13785.758,E2 -13785.758} C_VEL
LIN {X 0,Y 351.303,Z 725.057,A -85,B 0,C 180,E1 -13787.012,E2 -13787.012} C_VEL
LIN {X 0,Y 352.377,Z 714.256,A -85,B 0,C 180,E1 -13788.007,E2 -13788.007} C_VEL
LIN {X 0,Y 353.378,Z 701.219,A -85,B 0,C 180,E1 -13788.93,E2 -13788.93} C_VEL
LIN {X 0,Y 354.219,Z 688.677,A -85,B 0,C 180,E1 -13789.561,E2 -13789.561} C_VEL
LIN {X 0,Y 354.78,Z 675.545,A -85,B 0,C 180,E1 -13789.981,E2 -13789.981} C_VEL
LIN {X 0,Y 355.884,Z 604.744,A -85,B 0,C 180,E1 -13791.413,E2 -13791.413} C_VEL
LIN {X 0,Y 350.573,Z 570.483,A -85,B 0,C 180,E1 -13792.474,E2 -13792.474} C_VEL
LIN {X 0,Y 351.549,Z 560.798,A -85,B 0,C 180,E1 -13794.823,E2 -13794.823} C_VEL
LIN {X 0,Y 350.022,Z 551.852,A -85,B 0,C 180,E1 -13797.179,E2 -13797.179} C_VEL
LIN {X 0,Y 347.811,Z 541.163,A -85,B 0,C 180,E1 -13800.152,E2 -13800.152} C_VEL
LIN {X 0,Y 347.742,Z 541.166,A -85,B 0,C 180,E1 -13804.463,E2 -13804.463} C_VEL
LIN {X 0,Y 347.775,Z 541.163,A -85,B 0,C 180,E1 -13807.989,E2 -13807.989} C_VEL
LIN {X 0,Y 347.748,Z 541.167,A -85,B 0,C 180,E1 -13811.829,E2 -13811.829} C_VEL
LIN {X 0,Y 347.765,Z 541.164,A -85,B 0,C 180,E1 -13815.016,E2 -13815.016} C_VEL
LIN {X 0,Y 347.764,Z 541.163,A -85,B 0,C 180,E1 -13818.393,E2 -13818.393} C_VEL
LIN {X 0,Y 347.771,Z 541.163,A -85,B 0,C 180,E1 -13822.01,E2 -13822.01} C_VEL
LIN {X 0,Y 347.739,Z 541.171,A -85,B 0,C 180,E1 -13825.535,E2 -13825.535} C_VEL
LIN {X 0,Y 347.758,Z 541.167,A -85,B 0,C 180,E1 -13829.653,E2 -13829.653} C_VEL
LIN {X 0,Y 347.846,Z 541.152,A -85,B 0,C 180,E1 -13832.744,E2 -13832.744} C_VEL
LIN {X 0,Y 347.779,Z 541.161,A -85,B 0,C 180,E1 -13836.161,E2 -13836.161} C_VEL
LIN {X 0,Y 347.804,Z 541.159,A -85,B 0,C 180,E1 -13839.909,E2 -13839.909} C_VEL
LIN {X 0,Y 347.859,Z 541.15,A -85,B 0,C 180,E1 -13842.359,E2 -13842.359} C_VEL
LIN {X 0,Y 347.89,Z 541.148,A -85,B 0,C 180,E1 -13845.971,E2 -13845.971} C_VEL
LIN {X 0,Y 347.921,Z 541.148,A -85,B 0,C 180,E1 -13849.525,E2 -13849.525} C_VEL
LIN {X 0,Y 348.086,Z 541.125,A -85,B 0,C 180,E1 -13853.042,E2 -13853.042} C_VEL
LIN {X 0,Y 348.2,Z 541.112,A -85,B 0,C 180,E1 -13857.687,E2 -13857.687} C_VEL
LIN {X 0,Y 348.338,Z 541.092,A -85,B 0,C 180,E1 -13860,E2 -13860} C_VEL
LIN {X 0,Y 348.201,Z 541.107,A -85,B 0,C 180,E1 -13862.314,E2 -13862.314} C_VEL
LIN {X 0,Y 348.085,Z 541.124,A -85,B 0,C 180,E1 -13866.958,E2 -13866.958} C_VEL
LIN {X 0,Y 347.921,Z 541.142,A -85,B 0,C 180,E1 -13870.475,E2 -13870.475} C_VEL
LIN {X 0,Y 347.892,Z 541.147,A -85,B 0,C 180,E1 -13874.15,E2 -13874.15} C_VEL
LIN {X 0,Y 347.884,Z 541.147,A -85,B 0,C 180,E1 -13878.291,E2 -13878.291} C_VEL
LIN {X 0,Y 347.783,Z 541.164,A -85,B 0,C 180,E1 -13881.636,E2 -13881.636} C_VEL
LIN {X 0,Y 347.807,Z 541.16,A -85,B 0,C 180,E1 -13885.109,E2 -13885.109} C_VEL
LIN {X 0,Y 347.807,Z 541.161,A -85,B 0,C 180,E1 -13887.695,E2 -13887.695} C_VEL
LIN {X 0,Y 347.759,Z 541.163,A -85,B 0,C 180,E1 -13890.347,E2 -13890.347} C_VEL
LIN {X 0,Y 347.74,Z 541.165,A -85,B 0,C 180,E1 -13894.465,E2 -13894.465} C_VEL
LIN {X 0,Y 347.773,Z 541.161,A -85,B 0,C 180,E1 -13897.99,E2 -13897.99} C_VEL
LIN {X 0,Y 347.748,Z 541.167,A -85,B 0,C 180,E1 -13901.831,E2 -13901.831} C_VEL
LIN {X 0,Y 347.795,Z 541.161,A -85,B 0,C 180,E1 -13905.013,E2 -13905.013} C_VEL
LIN {X 0,Y 347.782,Z 541.16,A -85,B 0,C 180,E1 -13908.392,E2 -13908.392} C_VEL
LIN {X 0,Y 347.776,Z 541.162,A -85,B 0,C 180,E1 -13912.012,E2 -13912.012} C_VEL
LIN {X 0,Y 347.744,Z 541.17,A -85,B 0,C 180,E1 -13915.537,E2 -13915.537} C_VEL
LIN {X 0,Y 347.764,Z 541.167,A -85,B 0,C 180,E1 -13919.654,E2 -13919.654} C_VEL
LIN {X 0,Y 347.853,Z 541.153,A -85,B 0,C 180,E1 -13922.745,E2 -13922.745} C_VEL
LIN {X 0,Y 347.79,Z 541.16,A -85,B 0,C 180,E1 -13926.163,E2 -13926.163} C_VEL
LIN {X 0,Y 347.834,Z 541.239,A -85,B 0,C 180,E1 -13928.154,E2 -13928.154} C_VEL
LIN {X 0,Y 350.012,Z 552.291,A -85,B 0,C 180,E1 -13931.517,E2 -13931.517} C_VEL
LIN {X 0,Y 350.128,Z 552.791,A -85,B 0,C 180,E1 -13931.593,E2 -13931.593} C_VEL
LIN {X 0,Y 352.821,Z 561.178,A -85,B 0,C 180,E1 -13931.94,E2 -13931.94} C_VEL
LIN {X 0,Y 356.359,Z 579.895,A -85,B 0,C 180,E1 -13932.549,E2 -13932.549} C_VEL
LIN {X 0,Y 354.961,Z 659.397,A -85,B 0,C 180,E1 -13934.166,E2 -13934.166} C_VEL
LIN {X 0,Y 354.434,Z 671.806,A -85,B 0,C 180,E1 -13934.621,E2 -13934.621} C_VEL
LIN {X 0,Y 353.682,Z 684.643,A -85,B 0,C 180,E1 -13935.324,E2 -13935.324} C_VEL
LIN {X 0,Y 352.758,Z 696.046,A -85,B 0,C 180,E1 -13936.168,E2 -13936.168} C_VEL
LIN {X 0,Y 351.762,Z 707.722,A -85,B 0,C 180,E1 -13937.305,E2 -13937.305} C_VEL
LIN {X 0,Y 350.607,Z 718.201,A -85,B 0,C 180,E1 -13938.583,E2 -13938.583} C_VEL
LIN {X 0,Y 349.618,Z 726.922,A -85,B 0,C 180,E1 -13939.896,E2 -13939.896} C_VEL
LIN {X 0,Y 348.879,Z 734.646,A -85,B 0,C 180,E1 -13941.31,E2 -13941.31} C_VEL
LIN {X 0,Y 347.931,Z 742.384,A -85,B 0,C 180,E1 -13943.039,E2 -13943.039} C_VEL
LIN {X 0,Y 347.39,Z 748.563,A -85,B 0,C 180,E1 -13944.777,E2 -13944.777} C_VEL
LIN {X 0,Y 346.755,Z 753.494,A -85,B 0,C 180,E1 -13946.514,E2 -13946.514} C_VEL
LIN {X 0,Y 346.494,Z 757.303,A -85,B 0,C 180,E1 -13948.257,E2 -13948.257} C_VEL
LIN {X 0,Y 346.242,Z 760.106,A -85,B 0,C 180,E1 -13950,E2 -13950} C_VEL
LIN {X 0,Y 346.173,Z 761.43,A -85,B 0,C 180,E1 -13951.163,E2 -13951.163} C_VEL
LIN {X 0,Y 346.148,Z 762.918,A -85,B 0,C 180,E1 -13953.492,E2 -13953.492} C_VEL
LIN {X 0,Y 346.168,Z 763.045,A -85,B 0,C 180,E1 -13954.658,E2 -13954.658} C_VEL
LIN {X 0,Y 346.199,Z 762.755,A -85,B 0,C 180,E1 -13955.885,E2 -13955.885} C_VEL
LIN {X 0,Y 346.325,Z 761.097,A -85,B 0,C 180,E1 -13958.166,E2 -13958.166} C_VEL
LIN {X 0,Y 346.46,Z 759.617,A -85,B 0,C 180,E1 -13959.339,E2 -13959.339} C_VEL
LIN {X 0,Y 346.798,Z 756.606,A -85,B 0,C 180,E1 -13961.1,E2 -13961.1} C_VEL
LIN {X 0,Y 347.275,Z 752.535,A -85,B 0,C 180,E1 -13962.862,E2 -13962.862} C_VEL
LIN {X 0,Y 348.093,Z 746.271,A -85,B 0,C 180,E1 -13964.917,E2 -13964.917} C_VEL
LIN {X 0,Y 349.085,Z 739.434,A -85,B 0,C 180,E1 -13966.671,E2 -13966.671} C_VEL
LIN {X 0,Y 350.111,Z 732.436,A -85,B 0,C 180,E1 -13968.128,E2 -13968.128} C_VEL
LIN {X 0,Y 351.239,Z 723.984,A -85,B 0,C 180,E1 -13969.581,E2 -13969.581} C_VEL
LIN {X 0,Y 352.497,Z 713.504,A -85,B 0,C 180,E1 -13971.031,E2 -13971.031} C_VEL
LIN {X 0,Y 353.912,Z 701.671,A -85,B 0,C 180,E1 -13972.32,E2 -13972.32} C_VEL
LIN {X 0,Y 355.124,Z 689.735,A -85,B 0,C 180,E1 -13973.316,E2 -13973.316} C_VEL
LIN {X 0,Y 355.956,Z 677.248,A -85,B 0,C 180,E1 -13974.107,E2 -13974.107} C_VEL
LIN {X 0,Y 356.751,Z 664.257,A -85,B 0,C 180,E1 -13974.671,E2 -13974.671} C_VEL
LIN {X 0,Y 357.218,Z 649.139,A -85,B 0,C 180,E1 -13975.049,E2 -13975.049} C_VEL
LIN {X 0,Y 357.836,Z 614.486,A -85,B 0,C 180,E1 -13975.749,E2 -13975.749} C_VEL
LIN {X 0,Y 357.326,Z 608.684,A -85,B 0,C 180,E1 -13975.909,E2 -13975.909} C_VEL
LIN {X 0,Y 352.544,Z 590.009,A -85,B 0,C 180,E1 -13976.66,E2 -13976.66} C_VEL
LIN {X 0,Y 352.049,Z 584.207,A -85,B 0,C 180,E1 -13976.824,E2 -13976.824} C_VEL
LIN {X 0,Y 351.777,Z 580.301,A -85,B 0,C 180,E1 -13976.93,E2 -13976.93} C_VEL
LIN {X 0,Y 348.668,Z 566.718,A -85,B 0,C 180,E1 -13977.469,E2 -13977.469} C_VEL
LIN {X 0,Y 343.096,Z 552.808,A -85,B 0,C 180,E1 -13978.258,E2 -13978.258} C_VEL
LIN {X 0,Y 340.714,Z 542.049,A -85,B 0,C 180,E1 -13981.798,E2 -13981.798} C_VEL
LIN {X 0,Y 340.718,Z 542.042,A -85,B 0,C 180,E1 -13985.278,E2 -13985.278} C_VEL
LIN {X 0,Y 340.717,Z 542.041,A -85,B 0,C 180,E1 -13988.387,E2 -13988.387} C_VEL
LIN {X 0,Y 340.724,Z 542.042,A -85,B 0,C 180,E1 -13991.303,E2 -13991.303} C_VEL
LIN {X 0,Y 340.736,Z 542.044,A -85,B 0,C 180,E1 -13994.529,E2 -13994.529} C_VEL
LIN {X 0,Y 340.731,Z 542.037,A -85,B 0,C 180,E1 -13997.947,E2 -13997.947} C_VEL
LIN {X 0,Y 340.737,Z 542.04,A -85,B 0,C 180,E1 -14001.773,E2 -14001.773} C_VEL
LIN {X 0,Y 340.718,Z 542.04,A -85,B 0,C 180,E1 -14005.595,E2 -14005.595} C_VEL
LIN {X 0,Y 340.699,Z 542.041,A -85,B 0,C 180,E1 -14008.955,E2 -14008.955} C_VEL
LIN {X 0,Y 340.774,Z 542.036,A -85,B 0,C 180,E1 -14012.473,E2 -14012.473} C_VEL
LIN {X 0,Y 340.75,Z 542.038,A -85,B 0,C 180,E1 -14015.638,E2 -14015.638} C_VEL
LIN {X 0,Y 340.746,Z 542.038,A -85,B 0,C 180,E1 -14019.474,E2 -14019.474} C_VEL
LIN {X 0,Y 340.851,Z 542.021,A -85,B 0,C 180,E1 -14021.984,E2 -14021.984} C_VEL
LIN {X 0,Y 340.863,Z 542.023,A -85,B 0,C 180,E1 -14025.705,E2 -14025.705} C_VEL
LIN {X 0,Y 340.863,Z 542.024,A -85,B 0,C 180,E1 -14029.306,E2 -14029.306} C_VEL
LIN {X 0,Y 341.052,Z 541.996,A -85,B 0,C 180,E1 -14032.898,E2 -14032.898} C_VEL
LIN {X 0,Y 341.163,Z 541.977,A -85,B 0,C 180,E1 -14037.639,E2 -14037.639} C_VEL
LIN {X 0,Y 341.309,Z 541.968,A -85,B 0,C 180,E1 -14040,E2 -14040} C_VEL
LIN {X 0,Y 341.162,Z 541.984,A -85,B 0,C 180,E1 -14042.361,E2 -14042.361} C_VEL
LIN {X 0,Y 341.052,Z 541.998,A -85,B 0,C 180,E1 -14047.102,E2 -14047.102} C_VEL
LIN {X 0,Y 340.863,Z 542.028,A -85,B 0,C 180,E1 -14050.694,E2 -14050.694} C_VEL
LIN {X 0,Y 340.856,Z 542.019,A -85,B 0,C 180,E1 -14054.325,E2 -14054.325} C_VEL
LIN {X 0,Y 340.831,Z 542.024,A -85,B 0,C 180,E1 -14058.467,E2 -14058.467} C_VEL
LIN {X 0,Y 340.711,Z 542.042,A -85,B 0,C 180,E1 -14061.842,E2 -14061.842} C_VEL
LIN {X 0,Y 340.766,Z 542.035,A -85,B 0,C 180,E1 -14065.665,E2 -14065.665} C_VEL
LIN {X 0,Y 340.736,Z 542.037,A -85,B 0,C 180,E1 -14068.32,E2 -14068.32} C_VEL
LIN {X 0,Y 340.698,Z 542.046,A -85,B 0,C 180,E1 -14071.045,E2 -14071.045} C_VEL
LIN {X 0,Y 340.713,Z 542.043,A -85,B 0,C 180,E1 -14075.279,E2 -14075.279} C_VEL
LIN {X 0,Y 340.713,Z 542.046,A -85,B 0,C 180,E1 -14078.388,E2 -14078.388} C_VEL
LIN {X 0,Y 340.729,Z 542.043,A -85,B 0,C 180,E1 -14082.053,E2 -14082.053} C_VEL
LIN {X 0,Y 340.68,Z 542.048,A -85,B 0,C 180,E1 -14085.462,E2 -14085.462} C_VEL
LIN {X 0,Y 340.683,Z 542.051,A -85,B 0,C 180,E1 -14088.691,E2 -14088.691} C_VEL
LIN {X 0,Y 340.731,Z 542.042,A -85,B 0,C 180,E1 -14091.773,E2 -14091.773} C_VEL
LIN {X 0,Y 340.721,Z 542.044,A -85,B 0,C 180,E1 -14095.596,E2 -14095.596} C_VEL
LIN {X 0,Y 340.709,Z 542.193,A -85,B 0,C 180,E1 -14098.012,E2 -14098.012} C_VEL
LIN {X 0,Y 343.199,Z 552.735,A -85,B 0,C 180,E1 -14101.178,E2 -14101.178} C_VEL
LIN {X 0,Y 345.329,Z 563.373,A -85,B 0,C 180,E1 -14104.207,E2 -14104.207} C_VEL
LIN {X 0,Y 345.376,Z 566.474,A -85,B 0,C 180,E1 -14105.025,E2 -14105.025} C_VEL
LIN {X 0,Y 344.931,Z 570.162,A -85,B 0,C 180,E1 -14105.953,E2 -14105.953} C_VEL
LIN {X 0,Y 350.648,Z 600.51,A -85,B 0,C 180,E1 -14107.075,E2 -14107.075} C_VEL
LIN {X 0,Y 351.587,Z 608.228,A -85,B 0,C 180,E1 -14107.314,E2 -14107.314} C_VEL
LIN {X 0,Y 350.075,Z 678.9,A -85,B 0,C 180,E1 -14108.788,E2 -14108.788} C_VEL
LIN {X 0,Y 349.317,Z 692.513,A -85,B 0,C 180,E1 -14109.309,E2 -14109.309} C_VEL
LIN {X 0,Y 348.208,Z 704.962,A -85,B 0,C 180,E1 -14110.011,E2 -14110.011} C_VEL
LIN {X 0,Y 347.034,Z 716.851,A -85,B 0,C 180,E1 -14110.941,E2 -14110.941} C_VEL
LIN {X 0,Y 345.571,Z 728.267,A -85,B 0,C 180,E1 -14112.086,E2 -14112.086} C_VEL
LIN {X 0,Y 344.234,Z 738.569,A -85,B 0,C 180,E1 -14113.392,E2 -14113.392} C_VEL
LIN {X 0,Y 342.988,Z 747.833,A -85,B 0,C 180,E1 -14114.856,E2 -14114.856} C_VEL
LIN {X 0,Y 341.947,Z 755.475,A -85,B 0,C 180,E1 -14116.329,E2 -14116.329} C_VEL
LIN {X 0,Y 340.808,Z 762.973,A -85,B 0,C 180,E1 -14118.1,E2 -14118.1} C_VEL
LIN {X 0,Y 340.078,Z 769.011,A -85,B 0,C 180,E1 -14119.883,E2 -14119.883} C_VEL
LIN {X 0,Y 339.544,Z 773.801,A -85,B 0,C 180,E1 -14121.669,E2 -14121.669} C_VEL
LIN {X 0,Y 339.196,Z 777.481,A -85,B 0,C 180,E1 -14123.457,E2 -14123.457} C_VEL
LIN {X 0,Y 339.076,Z 780.155,A -85,B 0,C 180,E1 -14125.244,E2 -14125.244} C_VEL
LIN {X 0,Y 339.071,Z 781.421,A -85,B 0,C 180,E1 -14126.435,E2 -14126.435} C_VEL
LIN {X 0,Y 338.998,Z 782.286,A -85,B 0,C 180,E1 -14127.624,E2 -14127.624} C_VEL
LIN {X 0,Y 339.018,Z 782.718,A -85,B 0,C 180,E1 -14128.812,E2 -14128.812} C_VEL
LIN {X 0,Y 339.068,Z 782.76,A -85,B 0,C 180,E1 -14130,E2 -14130} C_VEL
LIN {X 0,Y 339.02,Z 782.414,A -85,B 0,C 180,E1 -14131.188,E2 -14131.188} C_VEL
LIN {X 0,Y 339,Z 781.679,A -85,B 0,C 180,E1 -14132.376,E2 -14132.376} C_VEL
LIN {X 0,Y 339.072,Z 780.503,A -85,B 0,C 180,E1 -14133.565,E2 -14133.565} C_VEL
LIN {X 0,Y 339.111,Z 777.072,A -85,B 0,C 180,E1 -14135.85,E2 -14135.85} C_VEL
LIN {X 0,Y 339.386,Z 772.986,A -85,B 0,C 180,E1 -14137.735,E2 -14137.735} C_VEL
LIN {X 0,Y 339.782,Z 767.938,A -85,B 0,C 180,E1 -14139.524,E2 -14139.524} C_VEL
LIN {X 0,Y 340.377,Z 761.589,A -85,B 0,C 180,E1 -14141.312,E2 -14141.312} C_VEL
LIN {X 0,Y 341.341,Z 753.635,A -85,B 0,C 180,E1 -14143.09,E2 -14143.09} C_VEL
LIN {X 0,Y 342.281,Z 745.525,A -85,B 0,C 180,E1 -14144.568,E2 -14144.568} C_VEL
LIN {X 0,Y 343.423,Z 734.869,A -85,B 0,C 180,E1 -14146.144,E2 -14146.144} C_VEL
LIN {X 0,Y 344.512,Z 724.529,A -85,B 0,C 180,E1 -14147.358,E2 -14147.358} C_VEL
LIN {X 0,Y 345.601,Z 713.648,A -85,B 0,C 180,E1 -14148.373,E2 -14148.373} C_VEL
LIN {X 0,Y 346.55,Z 701.633,A -85,B 0,C 180,E1 -14149.241,E2 -14149.241} C_VEL
LIN {X 0,Y 347.47,Z 688.555,A -85,B 0,C 180,E1 -14149.918,E2 -14149.918} C_VEL
LIN {X 0,Y 348.036,Z 675.686,A -85,B 0,C 180,E1 -14150.341,E2 -14150.341} C_VEL
LIN {X 0,Y 349.259,Z 605.908,A -85,B 0,C 180,E1 -14151.775,E2 -14151.775} C_VEL
LIN {X 0,Y 343.738,Z 570.338,A -85,B 0,C 180,E1 -14152.893,E2 -14152.893} C_VEL
LIN {X 0,Y 344.567,Z 561.703,A -85,B 0,C 180,E1 -14155.038,E2 -14155.038} C_VEL
LIN {X 0,Y 342.985,Z 552.757,A -85,B 0,C 180,E1 -14157.454,E2 -14157.454} C_VEL
LIN {X 0,Y 340.74,Z 542.044,A -85,B 0,C 180,E1 -14160.505,E2 -14160.505} C_VEL
LIN {X 0,Y 340.721,Z 542.041,A -85,B 0,C 180,E1 -14164.404,E2 -14164.404} C_VEL
LIN {X 0,Y 340.709,Z 542.042,A -85,B 0,C 180,E1 -14168.386,E2 -14168.386} C_VEL
LIN {X 0,Y 340.696,Z 542.044,A -85,B 0,C 180,E1 -14172.045,E2 -14172.045} C_VEL
LIN {X 0,Y 340.694,Z 542.049,A -85,B 0,C 180,E1 -14175.463,E2 -14175.463} C_VEL
LIN {X 0,Y 340.7,Z 542.043,A -85,B 0,C 180,E1 -14178.692,E2 -14178.692} C_VEL
LIN {X 0,Y 340.734,Z 542.041,A -85,B 0,C 180,E1 -14181.773,E2 -14181.773} C_VEL
LIN {X 0,Y 340.717,Z 542.045,A -85,B 0,C 180,E1 -14185.595,E2 -14185.595} C_VEL
LIN {X 0,Y 340.698,Z 542.044,A -85,B 0,C 180,E1 -14188.955,E2 -14188.955} C_VEL
LIN {X 0,Y 340.773,Z 542.033,A -85,B 0,C 180,E1 -14192.473,E2 -14192.473} C_VEL
LIN {X 0,Y 340.748,Z 542.04,A -85,B 0,C 180,E1 -14195.638,E2 -14195.638} C_VEL
LIN {X 0,Y 340.731,Z 542.045,A -85,B 0,C 180,E1 -14199.473,E2 -14199.473} C_VEL
LIN {X 0,Y 340.851,Z 542.024,A -85,B 0,C 180,E1 -14201.984,E2 -14201.984} C_VEL
LIN {X 0,Y 340.862,Z 542.026,A -85,B 0,C 180,E1 -14205.705,E2 -14205.705} C_VEL
LIN {X 0,Y 340.863,Z 542.026,A -85,B 0,C 180,E1 -14209.306,E2 -14209.306} C_VEL
LIN {X 0,Y 341.054,Z 542,A -85,B 0,C 180,E1 -14212.898,E2 -14212.898} C_VEL
LIN {X 0,Y 341.162,Z 541.989,A -85,B 0,C 180,E1 -14217.639,E2 -14217.639} C_VEL
LIN {X 0,Y 341.288,Z 541.97,A -85,B 0,C 180,E1 -14220,E2 -14220} C_VEL
LIN {X 0,Y 341.163,Z 541.983,A -85,B 0,C 180,E1 -14222.361,E2 -14222.361} C_VEL
LIN {X 0,Y 341.053,Z 542.001,A -85,B 0,C 180,E1 -14227.102,E2 -14227.102} C_VEL
LIN {X 0,Y 340.864,Z 542.02,A -85,B 0,C 180,E1 -14230.694,E2 -14230.694} C_VEL
LIN {X 0,Y 340.856,Z 542.023,A -85,B 0,C 180,E1 -14234.325,E2 -14234.325} C_VEL
LIN {X 0,Y 340.83,Z 542.025,A -85,B 0,C 180,E1 -14238.467,E2 -14238.467} C_VEL
LIN {X 0,Y 340.748,Z 542.038,A -85,B 0,C 180,E1 -14241.858,E2 -14241.858} C_VEL
LIN {X 0,Y 340.767,Z 542.037,A -85,B 0,C 180,E1 -14245.665,E2 -14245.665} C_VEL
LIN {X 0,Y 340.737,Z 542.038,A -85,B 0,C 180,E1 -14248.32,E2 -14248.32} C_VEL
LIN {X 0,Y 340.699,Z 542.045,A -85,B 0,C 180,E1 -14251.045,E2 -14251.045} C_VEL
LIN {X 0,Y 340.714,Z 542.046,A -85,B 0,C 180,E1 -14255.28,E2 -14255.28} C_VEL
LIN {X 0,Y 340.708,Z 542.04,A -85,B 0,C 180,E1 -14258.387,E2 -14258.387} C_VEL
LIN {X 0,Y 340.697,Z 542.044,A -85,B 0,C 180,E1 -14262.047,E2 -14262.047} C_VEL
LIN {X 0,Y 340.735,Z 542.043,A -85,B 0,C 180,E1 -14265.471,E2 -14265.471} C_VEL
LIN {X 0,Y 340.724,Z 542.04,A -85,B 0,C 180,E1 -14268.697,E2 -14268.697} C_VEL
LIN {X 0,Y 340.738,Z 542.04,A -85,B 0,C 180,E1 -14271.774,E2 -14271.774} C_VEL
LIN {X 0,Y 340.723,Z 542.044,A -85,B 0,C 180,E1 -14275.596,E2 -14275.596} C_VEL
LIN {X 0,Y 340.704,Z 542.045,A -85,B 0,C 180,E1 -14278.957,E2 -14278.957} C_VEL
LIN {X 0,Y 340.78,Z 542.033,A -85,B 0,C 180,E1 -14282.475,E2 -14282.475} C_VEL
LIN {X 0,Y 340.758,Z 542.039,A -85,B 0,C 180,E1 -14285.639,E2 -14285.639} C_VEL
LIN {X 0,Y 340.781,Z 542.144,A -85,B 0,C 180,E1 -14287.836,E2 -14287.836} C_VEL
LIN {X 0,Y 342.973,Z 552.938,A -85,B 0,C 180,E1 -14291.137,E2 -14291.137} C_VEL
LIN {X 0,Y 346.372,Z 563.14,A -85,B 0,C 180,E1 -14291.58,E2 -14291.58} C_VEL
LIN {X 0,Y 349.687,Z 580.663,A -85,B 0,C 180,E1 -14292.165,E2 -14292.165} C_VEL
LIN {X 0,Y 348.236,Z 660.014,A -85,B 0,C 180,E1 -14293.814,E2 -14293.814} C_VEL
LIN {X 0,Y 347.655,Z 673.042,A -85,B 0,C 180,E1 -14294.313,E2 -14294.313} C_VEL
LIN {X 0,Y 346.858,Z 685.616,A -85,B 0,C 180,E1 -14295.029,E2 -14295.029} C_VEL
LIN {X 0,Y 345.913,Z 696.812,A -85,B 0,C 180,E1 -14295.889,E2 -14295.889} C_VEL
LIN {X 0,Y 344.883,Z 708.366,A -85,B 0,C 180,E1 -14297.047,E2 -14297.047} C_VEL
LIN {X 0,Y 343.696,Z 718.769,A -85,B 0,C 180,E1 -14298.351,E2 -14298.351} C_VEL
LIN {X 0,Y 342.657,Z 727.628,A -85,B 0,C 180,E1 -14299.722,E2 -14299.722} C_VEL
LIN {X 0,Y 341.897,Z 735.104,A -85,B 0,C 180,E1 -14301.132,E2 -14301.132} C_VEL
LIN {X 0,Y 340.915,Z 742.779,A -85,B 0,C 180,E1 -14302.895,E2 -14302.895} C_VEL
LIN {X 0,Y 340.345,Z 748.922,A -85,B 0,C 180,E1 -14304.668,E2 -14304.668} C_VEL
LIN {X 0,Y 339.676,Z 753.821,A -85,B 0,C 180,E1 -14306.441,E2 -14306.441} C_VEL
LIN {X 0,Y 339.427,Z 757.598,A -85,B 0,C 180,E1 -14308.22,E2 -14308.22} C_VEL
LIN {X 0,Y 339.146,Z 760.373,A -85,B 0,C 180,E1 -14310,E2 -14310} C_VEL
LIN {X 0,Y 339.033,Z 762.605,A -85,B 0,C 180,E1 -14312.376,E2 -14312.376} C_VEL
LIN {X 0,Y 339.072,Z 763.137,A -85,B 0,C 180,E1 -14313.565,E2 -14313.565} C_VEL
LIN {X 0,Y 339.114,Z 762.964,A -85,B 0,C 180,E1 -14315.948,E2 -14315.948} C_VEL
LIN {X 0,Y 339.248,Z 761.25,A -85,B 0,C 180,E1 -14318.338,E2 -14318.338} C_VEL
LIN {X 0,Y 339.387,Z 759.745,A -85,B 0,C 180,E1 -14319.536,E2 -14319.536} C_VEL
LIN {X 0,Y 339.769,Z 756.704,A -85,B 0,C 180,E1 -14321.332,E2 -14321.332} C_VEL
LIN {X 0,Y 340.284,Z 752.601,A -85,B 0,C 180,E1 -14323.131,E2 -14323.131} C_VEL
LIN {X 0,Y 341.157,Z 746.303,A -85,B 0,C 180,E1 -14325.227,E2 -14325.227} C_VEL
LIN {X 0,Y 342.234,Z 739.427,A -85,B 0,C 180,E1 -14327.015,E2 -14327.015} C_VEL
LIN {X 0,Y 343.298,Z 732.385,A -85,B 0,C 180,E1 -14328.5,E2 -14328.5} C_VEL
LIN {X 0,Y 344.55,Z 723.225,A -85,B 0,C 180,E1 -14330.079,E2 -14330.079} C_VEL
LIN {X 0,Y 345.993,Z 712.127,A -85,B 0,C 180,E1 -14331.602,E2 -14331.602} C_VEL
LIN {X 0,Y 347.292,Z 701.366,A -85,B 0,C 180,E1 -14332.769,E2 -14332.769} C_VEL
LIN {X 0,Y 348.571,Z 689.258,A -85,B 0,C 180,E1 -14333.781,E2 -14333.781} C_VEL
LIN {X 0,Y 349.455,Z 676.56,A -85,B 0,C 180,E1 -14334.585,E2 -14334.585} C_VEL
LIN {X 0,Y 350.243,Z 663.878,A -85,B 0,C 180,E1 -14335.127,E2 -14335.127} C_VEL
LIN {X 0,Y 350.708,Z 648.819,A -85,B 0,C 180,E1 -14335.505,E2 -14335.505} C_VEL
LIN {X 0,Y 352.049,Z 584.207,A -85,B 0,C 180,E1 -14336.824,E2 -14336.824} C_VEL
LIN {X 0,Y 351.618,Z 580.41,A -85,B 0,C 180,E1 -14336.94,E2 -14336.94} C_VEL
LIN {X 0,Y 349.605,Z 575.13,A -85,B 0,C 180,E1 -14337.209,E2 -14337.209} C_VEL
LIN {X 0,Y 346.623,Z 570.383,A -85,B 0,C 180,E1 -14337.546,E2 -14337.546} C_VEL
LIN {X 0,Y 339.729,Z 561.063,A -85,B 0,C 180,E1 -14338.313,E2 -14338.313} C_VEL
LIN {X 0,Y 337.81,Z 557.675,A -85,B 0,C 180,E1 -14338.552,E2 -14338.552} C_VEL
LIN {X 0,Y 335.918,Z 553.05,A -85,B 0,C 180,E1 -14338.848,E2 -14338.848} C_VEL
LIN {X 0,Y 333.661,Z 542.934,A -85,B 0,C 180,E1 -14342.264,E2 -14342.264} C_VEL
LIN {X 0,Y 333.676,Z 542.923,A -85,B 0,C 180,E1 -14346.138,E2 -14346.138} C_VEL
LIN {X 0,Y 333.683,Z 542.922,A -85,B 0,C 180,E1 -14349.186,E2 -14349.186} C_VEL
LIN {X 0,Y 333.688,Z 542.921,A -85,B 0,C 180,E1 -14352.51,E2 -14352.51} C_VEL
LIN {X 0,Y 333.657,Z 542.921,A -85,B 0,C 180,E1 -14355.965,E2 -14355.965} C_VEL
LIN {X 0,Y 333.653,Z 542.911,A -85,B 0,C 180,E1 -14359.313,E2 -14359.313} C_VEL
LIN {X 0,Y 333.653,Z 542.924,A -85,B 0,C 180,E1 -14362.349,E2 -14362.349} C_VEL
LIN {X 0,Y 333.67,Z 542.919,A -85,B 0,C 180,E1 -14365.34,E2 -14365.34} C_VEL
LIN {X 0,Y 333.698,Z 542.91,A -85,B 0,C 180,E1 -14369.709,E2 -14369.709} C_VEL
LIN {X 0,Y 333.739,Z 542.913,A -85,B 0,C 180,E1 -14372.4,E2 -14372.4} C_VEL
LIN {X 0,Y 333.721,Z 542.915,A -85,B 0,C 180,E1 -14375.09,E2 -14375.09} C_VEL
LIN {X 0,Y 333.679,Z 542.921,A -85,B 0,C 180,E1 -14379.019,E2 -14379.019} C_VEL
LIN {X 0,Y 333.787,Z 542.901,A -85,B 0,C 180,E1 -14381.589,E2 -14381.589} C_VEL
LIN {X 0,Y 333.802,Z 542.902,A -85,B 0,C 180,E1 -14385.576,E2 -14385.576} C_VEL
LIN {X 0,Y 333.826,Z 542.902,A -85,B 0,C 180,E1 -14389.078,E2 -14389.078} C_VEL
LIN {X 0,Y 333.999,Z 542.873,A -85,B 0,C 180,E1 -14392.747,E2 -14392.747} C_VEL
LIN {X 0,Y 333.805,Z 542.904,A -85,B 0,C 180,E1 -14395.169,E2 -14395.169} C_VEL
LIN {X 0,Y 334.1,Z 542.857,A -85,B 0,C 180,E1 -14397.589,E2 -14397.589} C_VEL
LIN {X 0,Y 334.26,Z 542.846,A -85,B 0,C 180,E1 -14400,E2 -14400} C_VEL
LIN {X 0,Y 334.099,Z 542.863,A -85,B 0,C 180,E1 -14402.411,E2 -14402.411} C_VEL
LIN {X 0,Y 334.007,Z 542.879,A -85,B 0,C 180,E1 -14406.039,E2 -14406.039} C_VEL
LIN {X 0,Y 333.951,Z 542.879,A -85,B 0,C 180,E1 -14408.471,E2 -14408.471} C_VEL
LIN {X 0,Y 333.784,Z 542.907,A -85,B 0,C 180,E1 -14412.155,E2 -14412.155} C_VEL
LIN {X 0,Y 333.77,Z 542.907,A -85,B 0,C 180,E1 -14415.886,E2 -14415.886} C_VEL
LIN {X 0,Y 333.79,Z 542.901,A -85,B 0,C 180,E1 -14418.655,E2 -14418.655} C_VEL
LIN {X 0,Y 333.65,Z 542.921,A -85,B 0,C 180,E1 -14422.281,E2 -14422.281} C_VEL
LIN {X 0,Y 333.729,Z 542.913,A -85,B 0,C 180,E1 -14426.247,E2 -14426.247} C_VEL
LIN {X 0,Y 333.706,Z 542.917,A -85,B 0,C 180,E1 -14428.973,E2 -14428.973} C_VEL
LIN {X 0,Y 333.638,Z 542.926,A -85,B 0,C 180,E1 -14432.588,E2 -14432.588} C_VEL
LIN {X 0,Y 333.671,Z 542.921,A -85,B 0,C 180,E1 -14436.14,E2 -14436.14} C_VEL
LIN {X 0,Y 333.668,Z 542.921,A -85,B 0,C 180,E1 -14439.189,E2 -14439.189} C_VEL
LIN {X 0,Y 333.671,Z 542.924,A -85,B 0,C 180,E1 -14442.509,E2 -14442.509} C_VEL
LIN {X 0,Y 333.617,Z 542.928,A -85,B 0,C 180,E1 -14445.96,E2 -14445.96} C_VEL
LIN {X 0,Y 333.644,Z 542.924,A -85,B 0,C 180,E1 -14449.316,E2 -14449.316} C_VEL
LIN {X 0,Y 333.663,Z 542.924,A -85,B 0,C 180,E1 -14453.168,E2 -14453.168} C_VEL
LIN {X 0,Y 333.672,Z 542.922,A -85,B 0,C 180,E1 -14455.342,E2 -14455.342} C_VEL
LIN {X 0,Y 333.677,Z 543.101,A -85,B 0,C 180,E1 -14457.527,E2 -14457.527} C_VEL
LIN {X 0,Y 336.041,Z 552.9,A -85,B 0,C 180,E1 -14460.563,E2 -14460.563} C_VEL
LIN {X 0,Y 338.141,Z 563.296,A -85,B 0,C 180,E1 -14463.611,E2 -14463.611} C_VEL
LIN {X 0,Y 338.606,Z 566.423,A -85,B 0,C 180,E1 -14464.49,E2 -14464.49} C_VEL
LIN {X 0,Y 338.22,Z 569.952,A -85,B 0,C 180,E1 -14465.403,E2 -14465.403} C_VEL
LIN {X 0,Y 343.777,Z 599.157,A -85,B 0,C 180,E1 -14466.525,E2 -14466.525} C_VEL
LIN {X 0,Y 345.114,Z 608.817,A -85,B 0,C 180,E1 -14466.845,E2 -14466.845} C_VEL
LIN {X 0,Y 343.532,Z 678.894,A -85,B 0,C 180,E1 -14468.334,E2 -14468.334} C_VEL
LIN {X 0,Y 342.755,Z 692.252,A -85,B 0,C 180,E1 -14468.854,E2 -14468.854} C_VEL
LIN {X 0,Y 341.628,Z 704.164,A -85,B 0,C 180,E1 -14469.53,E2 -14469.53} C_VEL
LIN {X 0,Y 340.546,Z 715.428,A -85,B 0,C 180,E1 -14470.406,E2 -14470.406} C_VEL
LIN {X 0,Y 339.015,Z 727.069,A -85,B 0,C 180,E1 -14471.571,E2 -14471.571} C_VEL
LIN {X 0,Y 337.582,Z 737.542,A -85,B 0,C 180,E1 -14472.899,E2 -14472.899} C_VEL
LIN {X 0,Y 336.356,Z 746.112,A -85,B 0,C 180,E1 -14474.239,E2 -14474.239} C_VEL
LIN {X 0,Y 335.265,Z 754.024,A -85,B 0,C 180,E1 -14475.741,E2 -14475.741} C_VEL
LIN {X 0,Y 334.012,Z 761.776,A -85,B 0,C 180,E1 -14477.545,E2 -14477.545} C_VEL
LIN {X 0,Y 333.061,Z 768.909,A -85,B 0,C 180,E1 -14479.668,E2 -14479.668} C_VEL
LIN {X 0,Y 332.493,Z 773.676,A -85,B 0,C 180,E1 -14481.491,E2 -14481.491} C_VEL
LIN {X 0,Y 332.12,Z 777.335,A -85,B 0,C 180,E1 -14483.317,E2 -14483.317} C_VEL
LIN {X 0,Y 331.981,Z 779.99,A -85,B 0,C 180,E1 -14485.143,E2 -14485.143} C_VEL
LIN {X 0,Y 331.996,Z 781.248,A -85,B 0,C 180,E1 -14486.359,E2 -14486.359} C_VEL
LIN {X 0,Y 331.916,Z 782.099,A -85,B 0,C 180,E1 -14487.573,E2 -14487.573} C_VEL
LIN {X 0,Y 331.923,Z 782.518,A -85,B 0,C 180,E1 -14488.787,E2 -14488.787} C_VEL
LIN {X 0,Y 331.971,Z 782.551,A -85,B 0,C 180,E1 -14490,E2 -14490} C_VEL
LIN {X 0,Y 331.925,Z 782.196,A -85,B 0,C 180,E1 -14491.213,E2 -14491.213} C_VEL
LIN {X 0,Y 331.918,Z 781.449,A -85,B 0,C 180,E1 -14492.427,E2 -14492.427} C_VEL
LIN {X 0,Y 331.997,Z 780.258,A -85,B 0,C 180,E1 -14493.641,E2 -14493.641} C_VEL
LIN {X 0,Y 332.009,Z 777.139,A -85,B 0,C 180,E1 -14495.787,E2 -14495.787} C_VEL
LIN {X 0,Y 332.326,Z 772.7,A -85,B 0,C 180,E1 -14497.901,E2 -14497.901} C_VEL
LIN {X 0,Y 332.757,Z 767.629,A -85,B 0,C 180,E1 -14499.727,E2 -14499.727} C_VEL
LIN {X 0,Y 333.378,Z 761.247,A -85,B 0,C 180,E1 -14501.553,E2 -14501.553} C_VEL
LIN {X 0,Y 334.416,Z 753.26,A -85,B 0,C 180,E1 -14503.366,E2 -14503.366} C_VEL
LIN {X 0,Y 335.385,Z 745.179,A -85,B 0,C 180,E1 -14504.863,E2 -14504.863} C_VEL
LIN {X 0,Y 336.44,Z 735.603,A -85,B 0,C 180,E1 -14506.317,E2 -14506.317} C_VEL
LIN {X 0,Y 337.563,Z 725.398,A -85,B 0,C 180,E1 -14507.571,E2 -14507.571} C_VEL
LIN {X 0,Y 338.694,Z 714.814,A -85,B 0,C 180,E1 -14508.604,E2 -14508.604} C_VEL
LIN {X 0,Y 339.749,Z 702.044,A -85,B 0,C 180,E1 -14509.563,E2 -14509.563} C_VEL
LIN {X 0,Y 340.661,Z 689.254,A -85,B 0,C 180,E1 -14510.255,E2 -14510.255} C_VEL
LIN {X 0,Y 341.32,Z 676.016,A -85,B 0,C 180,E1 -14510.709,E2 -14510.709} C_VEL
LIN {X 0,Y 342.49,Z 606.033,A -85,B 0,C 180,E1 -14512.184,E2 -14512.184} C_VEL
LIN {X 0,Y 337.254,Z 572.289,A -85,B 0,C 180,E1 -14513.268,E2 -14513.268} C_VEL
LIN {X 0,Y 336.912,Z 570.115,A -85,B 0,C 180,E1 -14513.349,E2 -14513.349} C_VEL
LIN {X 0,Y 337.585,Z 562.597,A -85,B 0,C 180,E1 -14515.263,E2 -14515.263} C_VEL
LIN {X 0,Y 335.533,Z 551.351,A -85,B 0,C 180,E1 -14518.391,E2 -14518.391} C_VEL
LIN {X 0,Y 333.678,Z 542.922,A -85,B 0,C 180,E1 -14520.888,E2 -14520.888} C_VEL
LIN {X 0,Y 333.684,Z 542.918,A -85,B 0,C 180,E1 -14524.773,E2 -14524.773} C_VEL
LIN {X 0,Y 333.652,Z 542.925,A -85,B 0,C 180,E1 -14527.65,E2 -14527.65} C_VEL
LIN {X 0,Y 333.644,Z 542.922,A -85,B 0,C 180,E1 -14530.767,E2 -14530.767} C_VEL
LIN {X 0,Y 333.622,Z 542.925,A -85,B 0,C 180,E1 -14534.255,E2 -14534.255} C_VEL
LIN {X 0,Y 333.677,Z 542.922,A -85,B 0,C 180,E1 -14537.624,E2 -14537.624} C_VEL
LIN {X 0,Y 333.673,Z 542.921,A -85,B 0,C 180,E1 -14541.196,E2 -14541.196} C_VEL
LIN {X 0,Y 333.68,Z 542.921,A -85,B 0,C 180,E1 -14545.225,E2 -14545.225} C_VEL
LIN {X 0,Y 333.692,Z 542.92,A -85,B 0,C 180,E1 -14549.637,E2 -14549.637} C_VEL
LIN {X 0,Y 333.738,Z 542.909,A -85,B 0,C 180,E1 -14552.401,E2 -14552.401} C_VEL
LIN {X 0,Y 333.719,Z 542.915,A -85,B 0,C 180,E1 -14555.09,E2 -14555.09} C_VEL
LIN {X 0,Y 333.668,Z 542.92,A -85,B 0,C 180,E1 -14559.018,E2 -14559.018} C_VEL
LIN {X 0,Y 333.787,Z 542.907,A -85,B 0,C 180,E1 -14561.589,E2 -14561.589} C_VEL
LIN {X 0,Y 333.801,Z 542.907,A -85,B 0,C 180,E1 -14565.576,E2 -14565.576} C_VEL
LIN {X 0,Y 333.826,Z 542.9,A -85,B 0,C 180,E1 -14569.078,E2 -14569.078} C_VEL
LIN {X 0,Y 334.006,Z 542.877,A -85,B 0,C 180,E1 -14572.747,E2 -14572.747} C_VEL
LIN {X 0,Y 333.804,Z 542.904,A -85,B 0,C 180,E1 -14575.169,E2 -14575.169} C_VEL
LIN {X 0,Y 334.099,Z 542.869,A -85,B 0,C 180,E1 -14577.589,E2 -14577.589} C_VEL
LIN {X 0,Y 334.239,Z 542.848,A -85,B 0,C 180,E1 -14580,E2 -14580} C_VEL
LIN {X 0,Y 334.1,Z 542.863,A -85,B 0,C 180,E1 -14582.411,E2 -14582.411} C_VEL
LIN {X 0,Y 333.986,Z 542.879,A -85,B 0,C 180,E1 -14586.647,E2 -14586.647} C_VEL
LIN {X 0,Y 333.843,Z 542.897,A -85,B 0,C 180,E1 -14589.696,E2 -14589.696} C_VEL
LIN {X 0,Y 333.789,Z 542.908,A -85,B 0,C 180,E1 -14593.392,E2 -14593.392} C_VEL
LIN {X 0,Y 333.74,Z 542.913,A -85,B 0,C 180,E1 -14597.147,E2 -14597.147} C_VEL
LIN {X 0,Y 333.73,Z 542.911,A -85,B 0,C 180,E1 -14599.691,E2 -14599.691} C_VEL
LIN {X 0,Y 333.687,Z 542.916,A -85,B 0,C 180,E1 -14602.279,E2 -14602.279} C_VEL
LIN {X 0,Y 333.73,Z 542.91,A -85,B 0,C 180,E1 -14606.247,E2 -14606.247} C_VEL
LIN {X 0,Y 333.706,Z 542.916,A -85,B 0,C 180,E1 -14608.973,E2 -14608.973} C_VEL
LIN {X 0,Y 333.639,Z 542.922,A -85,B 0,C 180,E1 -14612.588,E2 -14612.588} C_VEL
LIN {X 0,Y 333.673,Z 542.917,A -85,B 0,C 180,E1 -14616.14,E2 -14616.14} C_VEL
LIN {X 0,Y 333.644,Z 542.923,A -85,B 0,C 180,E1 -14619.193,E2 -14619.193} C_VEL
LIN {X 0,Y 333.632,Z 542.923,A -85,B 0,C 180,E1 -14622.501,E2 -14622.501} C_VEL
LIN {X 0,Y 333.672,Z 542.919,A -85,B 0,C 180,E1 -14625.969,E2 -14625.969} C_VEL
LIN {X 0,Y 333.7,Z 542.919,A -85,B 0,C 180,E1 -14629.305,E2 -14629.305} C_VEL
LIN {X 0,Y 333.665,Z 542.923,A -85,B 0,C 180,E1 -14633.168,E2 -14633.168} C_VEL
LIN {X 0,Y 333.674,Z 542.924,A -85,B 0,C 180,E1 -14635.342,E2 -14635.342} C_VEL
LIN {X 0,Y 333.703,Z 542.918,A -85,B 0,C 180,E1 -14639.711,E2 -14639.711} C_VEL
LIN {X 0,Y 333.744,Z 542.91,A -85,B 0,C 180,E1 -14642.402,E2 -14642.402} C_VEL
LIN {X 0,Y 333.728,Z 542.914,A -85,B 0,C 180,E1 -14645.091,E2 -14645.091} C_VEL
LIN {X 0,Y 333.717,Z 542.987,A -85,B 0,C 180,E1 -14647.479,E2 -14647.479} C_VEL
LIN {X 0,Y 335.746,Z 552.864,A -85,B 0,C 180,E1 -14650.631,E2 -14650.631} C_VEL
LIN {X 0,Y 340.034,Z 565.584,A -85,B 0,C 180,E1 -14651.223,E2 -14651.223} C_VEL
LIN {X 0,Y 343.002,Z 582.328,A -85,B 0,C 180,E1 -14651.785,E2 -14651.785} C_VEL
LIN {X 0,Y 341.554,Z 659.486,A -85,B 0,C 180,E1 -14653.412,E2 -14653.412} C_VEL
LIN {X 0,Y 341.002,Z 672.003,A -85,B 0,C 180,E1 -14653.884,E2 -14653.884} C_VEL
LIN {X 0,Y 340.224,Z 684.336,A -85,B 0,C 180,E1 -14654.576,E2 -14654.576} C_VEL
LIN {X 0,Y 339.225,Z 695.902,A -85,B 0,C 180,E1 -14655.452,E2 -14655.452} C_VEL
LIN {X 0,Y 338.162,Z 707.723,A -85,B 0,C 180,E1 -14656.632,E2 -14656.632} C_VEL
LIN {X 0,Y 336.913,Z 718.272,A -85,B 0,C 180,E1 -14657.96,E2 -14657.96} C_VEL
LIN {X 0,Y 335.76,Z 727.205,A -85,B 0,C 180,E1 -14659.347,E2 -14659.347} C_VEL
LIN {X 0,Y 334.904,Z 735.677,A -85,B 0,C 180,E1 -14660.97,E2 -14660.97} C_VEL
LIN {X 0,Y 333.901,Z 743.172,A -85,B 0,C 180,E1 -14662.745,E2 -14662.745} C_VEL
LIN {X 0,Y 333.283,Z 749.28,A -85,B 0,C 180,E1 -14664.555,E2 -14664.555} C_VEL
LIN {X 0,Y 332.599,Z 754.147,A -85,B 0,C 180,E1 -14666.366,E2 -14666.366} C_VEL
LIN {X 0,Y 332.361,Z 757.893,A -85,B 0,C 180,E1 -14668.182,E2 -14668.182} C_VEL
LIN {X 0,Y 332.049,Z 760.64,A -85,B 0,C 180,E1 -14670,E2 -14670} C_VEL
LIN {X 0,Y 331.948,Z 762.844,A -85,B 0,C 180,E1 -14672.427,E2 -14672.427} C_VEL
LIN {X 0,Y 331.997,Z 763.353,A -85,B 0,C 180,E1 -14673.641,E2 -14673.641} C_VEL
LIN {X 0,Y 332.033,Z 763.148,A -85,B 0,C 180,E1 -14676.075,E2 -14676.075} C_VEL
LIN {X 0,Y 332.063,Z 762.474,A -85,B 0,C 180,E1 -14677.295,E2 -14677.295} C_VEL
LIN {X 0,Y 332.187,Z 761.399,A -85,B 0,C 180,E1 -14678.516,E2 -14678.516} C_VEL
LIN {X 0,Y 332.326,Z 759.875,A -85,B 0,C 180,E1 -14679.74,E2 -14679.74} C_VEL
LIN {X 0,Y 332.748,Z 756.804,A -85,B 0,C 180,E1 -14681.575,E2 -14681.575} C_VEL
LIN {X 0,Y 333.311,Z 752.668,A -85,B 0,C 180,E1 -14683.411,E2 -14683.411} C_VEL
LIN {X 0,Y 334.247,Z 746.336,A -85,B 0,C 180,E1 -14685.55,E2 -14685.55} C_VEL
LIN {X 0,Y 335.371,Z 739.419,A -85,B 0,C 180,E1 -14687.374,E2 -14687.374} C_VEL
LIN {X 0,Y 336.521,Z 732.333,A -85,B 0,C 180,E1 -14688.887,E2 -14688.887} C_VEL
LIN {X 0,Y 337.725,Z 723.839,A -85,B 0,C 180,E1 -14690.382,E2 -14690.382} C_VEL
LIN {X 0,Y 339.179,Z 713.11,A -85,B 0,C 180,E1 -14691.898,E2 -14691.898} C_VEL
LIN {X 0,Y 340.533,Z 702.539,A -85,B 0,C 180,E1 -14693.086,E2 -14693.086} C_VEL
LIN {X 0,Y 341.863,Z 690.785,A -85,B 0,C 180,E1 -14694.116,E2 -14694.116} C_VEL
LIN {X 0,Y 342.755,Z 678.496,A -85,B 0,C 180,E1 -14694.936,E2 -14694.936} C_VEL
LIN {X 0,Y 343.666,Z 665.038,A -85,B 0,C 180,E1 -14695.552,E2 -14695.552} C_VEL
LIN {X 0,Y 344.138,Z 651.069,A -85,B 0,C 180,E1 -14695.927,E2 -14695.927} C_VEL
LIN {X 0,Y 345.546,Z 582.487,A -85,B 0,C 180,E1 -14697.358,E2 -14697.358} C_VEL
LIN {X 0,Y 342.672,Z 569.607,A -85,B 0,C 180,E1 -14697.877,E2 -14697.877} C_VEL
LIN {X 0,Y 337.81,Z 557.675,A -85,B 0,C 180,E1 -14698.552,E2 -14698.552} C_VEL
LIN {X 0,Y 335.786,Z 554.783,A -85,B 0,C 180,E1 -14698.863,E2 -14698.863} C_VEL
LIN {X 0,Y 333.412,Z 552.759,A -85,B 0,C 180,E1 -14699.306,E2 -14699.306} C_VEL
LIN {X 0,Y 330.369,Z 550.998,A -85,B 0,C 180,E1 -14700.032,E2 -14700.032} C_VEL
LIN {X 0,Y 328.117,Z 549.13,A -85,B 0,C 180,E1 -14700.865,E2 -14700.865} C_VEL
LIN {X 0,Y 327.572,Z 547.95,A -85,B 0,C 180,E1 -14701.298,E2 -14701.298} C_VEL
LIN {X 0,Y 326.604,Z 543.802,A -85,B 0,C 180,E1 -14702.829,E2 -14702.829} C_VEL
LIN {X 0,Y 326.612,Z 543.8,A -85,B 0,C 180,E1 -14705.519,E2 -14705.519} C_VEL
LIN {X 0,Y 326.644,Z 543.799,A -85,B 0,C 180,E1 -14709.233,E2 -14709.233} C_VEL
LIN {X 0,Y 326.627,Z 543.799,A -85,B 0,C 180,E1 -14712.981,E2 -14712.981} C_VEL
LIN {X 0,Y 326.614,Z 543.799,A -85,B 0,C 180,E1 -14717.019,E2 -14717.019} C_VEL
LIN {X 0,Y 326.64,Z 543.797,A -85,B 0,C 180,E1 -14721.393,E2 -14721.393} C_VEL
LIN {X 0,Y 326.616,Z 543.801,A -85,B 0,C 180,E1 -14724.85,E2 -14724.85} C_VEL
LIN {X 0,Y 326.603,Z 543.801,A -85,B 0,C 180,E1 -14727.455,E2 -14727.455} C_VEL
LIN {X 0,Y 326.656,Z 543.79,A -85,B 0,C 180,E1 -14730.34,E2 -14730.34} C_VEL
LIN {X 0,Y 326.685,Z 543.788,A -85,B 0,C 180,E1 -14734.516,E2 -14734.516} C_VEL
LIN {X 0,Y 326.642,Z 543.792,A -85,B 0,C 180,E1 -14738.545,E2 -14738.545} C_VEL
LIN {X 0,Y 326.738,Z 543.78,A -85,B 0,C 180,E1 -14741.177,E2 -14741.177} C_VEL
LIN {X 0,Y 326.756,Z 543.78,A -85,B 0,C 180,E1 -14745.433,E2 -14745.433} C_VEL
LIN {X 0,Y 326.762,Z 543.782,A -85,B 0,C 180,E1 -14748.838,E2 -14748.838} C_VEL
LIN {X 0,Y 326.951,Z 543.75,A -85,B 0,C 180,E1 -14752.59,E2 -14752.59} C_VEL
LIN {X 0,Y 326.771,Z 543.781,A -85,B 0,C 180,E1 -14755.065,E2 -14755.065} C_VEL
LIN {X 0,Y 327.041,Z 543.736,A -85,B 0,C 180,E1 -14757.537,E2 -14757.537} C_VEL
LIN {X 0,Y 327.21,Z 543.724,A -85,B 0,C 180,E1 -14760,E2 -14760} C_VEL
LIN {X 0,Y 327.04,Z 543.741,A -85,B 0,C 180,E1 -14762.463,E2 -14762.463} C_VEL
LIN {X 0,Y 326.982,Z 543.755,A -85,B 0,C 180,E1 -14766.169,E2 -14766.169} C_VEL
LIN {X 0,Y 326.798,Z 543.772,A -85,B 0,C 180,E1 -14769.907,E2 -14769.907} C_VEL
LIN {X 0,Y 326.752,Z 543.772,A -85,B 0,C 180,E1 -14773.686,E2 -14773.686} C_VEL
LIN {X 0,Y 326.692,Z 543.785,A -85,B 0,C 180,E1 -14777.528,E2 -14777.528} C_VEL
LIN {X 0,Y 326.653,Z 543.794,A -85,B 0,C 180,E1 -14780.136,E2 -14780.136} C_VEL
LIN {X 0,Y 326.642,Z 543.792,A -85,B 0,C 180,E1 -14784.13,E2 -14784.13} C_VEL
LIN {X 0,Y 326.679,Z 543.785,A -85,B 0,C 180,E1 -14786.858,E2 -14786.858} C_VEL
LIN {X 0,Y 326.633,Z 543.798,A -85,B 0,C 180,E1 -14790.612,E2 -14790.612} C_VEL
LIN {X 0,Y 326.602,Z 543.801,A -85,B 0,C 180,E1 -14794.02,E2 -14794.02} C_VEL
LIN {X 0,Y 326.625,Z 543.798,A -85,B 0,C 180,E1 -14797.24,E2 -14797.24} C_VEL
LIN {X 0,Y 326.6,Z 543.803,A -85,B 0,C 180,E1 -14800.208,E2 -14800.208} C_VEL
LIN {X 0,Y 326.599,Z 543.803,A -85,B 0,C 180,E1 -14803.519,E2 -14803.519} C_VEL
LIN {X 0,Y 326.578,Z 543.806,A -85,B 0,C 180,E1 -14807.028,E2 -14807.028} C_VEL
LIN {X 0,Y 326.609,Z 543.803,A -85,B 0,C 180,E1 -14810.774,E2 -14810.774} C_VEL
LIN {X 0,Y 326.61,Z 543.799,A -85,B 0,C 180,E1 -14814.481,E2 -14814.481} C_VEL
LIN {X 0,Y 326.615,Z 543.816,A -85,B 0,C 180,E1 -14816.959,E2 -14816.959} C_VEL
LIN {X 0,Y 329.335,Z 555.319,A -85,B 0,C 180,E1 -14820.606,E2 -14820.606} C_VEL
LIN {X 0,Y 331.291,Z 565.131,A -85,B 0,C 180,E1 -14823.546,E2 -14823.546} C_VEL
LIN {X 0,Y 331.638,Z 568.814,A -85,B 0,C 180,E1 -14824.588,E2 -14824.588} C_VEL
LIN {X 0,Y 331.532,Z 569.735,A -85,B 0,C 180,E1 -14824.831,E2 -14824.831} C_VEL
LIN {X 0,Y 336.94,Z 597.823,A -85,B 0,C 180,E1 -14825.952,E2 -14825.952} C_VEL
LIN {X 0,Y 338.673,Z 609.162,A -85,B 0,C 180,E1 -14826.353,E2 -14826.353} C_VEL
LIN {X 0,Y 337.061,Z 678.026,A -85,B 0,C 180,E1 -14827.835,E2 -14827.835} C_VEL
LIN {X 0,Y 336.237,Z 691.239,A -85,B 0,C 180,E1 -14828.344,E2 -14828.344} C_VEL
LIN {X 0,Y 335.007,Z 704.476,A -85,B 0,C 180,E1 -14829.107,E2 -14829.107} C_VEL
LIN {X 0,Y 333.866,Z 715.593,A -85,B 0,C 180,E1 -14829.998,E2 -14829.998} C_VEL
LIN {X 0,Y 332.275,Z 727.163,A -85,B 0,C 180,E1 -14831.183,E2 -14831.183} C_VEL
LIN {X 0,Y 330.776,Z 737.585,A -85,B 0,C 180,E1 -14832.536,E2 -14832.536} C_VEL
LIN {X 0,Y 329.518,Z 746.113,A -85,B 0,C 180,E1 -14833.903,E2 -14833.903} C_VEL
LIN {X 0,Y 328.374,Z 753.991,A -85,B 0,C 180,E1 -14835.435,E2 -14835.435} C_VEL
LIN {X 0,Y 327.055,Z 761.699,A -85,B 0,C 180,E1 -14837.276,E2 -14837.276} C_VEL
LIN {X 0,Y 326.058,Z 768.808,A -85,B 0,C 180,E1 -14839.443,E2 -14839.443} C_VEL
LIN {X 0,Y 325.457,Z 773.552,A -85,B 0,C 180,E1 -14841.306,E2 -14841.306} C_VEL
LIN {X 0,Y 325.06,Z 777.191,A -85,B 0,C 180,E1 -14843.171,E2 -14843.171} C_VEL
LIN {X 0,Y 324.892,Z 779.826,A -85,B 0,C 180,E1 -14845.036,E2 -14845.036} C_VEL
LIN {X 0,Y 324.9,Z 781.076,A -85,B 0,C 180,E1 -14846.279,E2 -14846.279} C_VEL
LIN {X 0,Y 324.836,Z 781.91,A -85,B 0,C 180,E1 -14847.52,E2 -14847.52} C_VEL
LIN {X 0,Y 324.875,Z 782.342,A -85,B 0,C 180,E1 -14850,E2 -14850} C_VEL
LIN {X 0,Y 324.833,Z 781.978,A -85,B 0,C 180,E1 -14851.24,E2 -14851.24} C_VEL
LIN {X 0,Y 324.838,Z 781.216,A -85,B 0,C 180,E1 -14852.48,E2 -14852.48} C_VEL
LIN {X 0,Y 324.901,Z 780.012,A -85,B 0,C 180,E1 -14853.721,E2 -14853.721} C_VEL
LIN {X 0,Y 324.914,Z 777.185,A -85,B 0,C 180,E1 -14855.733,E2 -14855.733} C_VEL
LIN {X 0,Y 325.256,Z 772.413,A -85,B 0,C 180,E1 -14858.074,E2 -14858.074} C_VEL
LIN {X 0,Y 325.814,Z 766.331,A -85,B 0,C 180,E1 -14860.251,E2 -14860.251} C_VEL
LIN {X 0,Y 326.524,Z 759.661,A -85,B 0,C 180,E1 -14862.114,E2 -14862.114} C_VEL
LIN {X 0,Y 327.688,Z 751.387,A -85,B 0,C 180,E1 -14863.962,E2 -14863.962} C_VEL
LIN {X 0,Y 328.816,Z 742.326,A -85,B 0,C 180,E1 -14865.592,E2 -14865.592} C_VEL
LIN {X 0,Y 329.897,Z 732.408,A -85,B 0,C 180,E1 -14867.033,E2 -14867.033} C_VEL
LIN {X 0,Y 331.204,Z 720.587,A -85,B 0,C 180,E1 -14868.399,E2 -14868.399} C_VEL
LIN {X 0,Y 332.455,Z 708.727,A -85,B 0,C 180,E1 -14869.447,E2 -14869.447} C_VEL
LIN {X 0,Y 333.471,Z 696.368,A -85,B 0,C 180,E1 -14870.268,E2 -14870.268} C_VEL
LIN {X 0,Y 334.276,Z 683.695,A -85,B 0,C 180,E1 -14870.861,E2 -14870.861} C_VEL
LIN {X 0,Y 334.72,Z 670.597,A -85,B 0,C 180,E1 -14871.232,E2 -14871.232} C_VEL
LIN {X 0,Y 335.859,Z 607.018,A -85,B 0,C 180,E1 -14872.581,E2 -14872.581} C_VEL
LIN {X 0,Y 330.657,Z 573.382,A -85,B 0,C 180,E1 -14873.692,E2 -14873.692} C_VEL
LIN {X 0,Y 330.052,Z 569.941,A -85,B 0,C 180,E1 -14873.816,E2 -14873.816} C_VEL
LIN {X 0,Y 330.684,Z 564.76,A -85,B 0,C 180,E1 -14875.154,E2 -14875.154} C_VEL
LIN {X 0,Y 329.443,Z 557.126,A -85,B 0,C 180,E1 -14877.3,E2 -14877.3} C_VEL
LIN {X 0,Y 327.402,Z 547.122,A -85,B 0,C 180,E1 -14880.224,E2 -14880.224} C_VEL
LIN {X 0,Y 326.628,Z 543.802,A -85,B 0,C 180,E1 -14881.271,E2 -14881.271} C_VEL
LIN {X 0,Y 326.618,Z 543.801,A -85,B 0,C 180,E1 -14885.148,E2 -14885.148} C_VEL
LIN {X 0,Y 326.622,Z 543.797,A -85,B 0,C 180,E1 -14888.608,E2 -14888.608} C_VEL
LIN {X 0,Y 326.573,Z 543.805,A -85,B 0,C 180,E1 -14891.845,E2 -14891.845} C_VEL
LIN {X 0,Y 326.567,Z 543.807,A -85,B 0,C 180,E1 -14895.249,E2 -14895.249} C_VEL
LIN {X 0,Y 326.589,Z 543.802,A -85,B 0,C 180,E1 -14898.865,E2 -14898.865} C_VEL
LIN {X 0,Y 326.638,Z 543.799,A -85,B 0,C 180,E1 -14901.393,E2 -14901.393} C_VEL
LIN {X 0,Y 326.614,Z 543.798,A -85,B 0,C 180,E1 -14904.851,E2 -14904.851} C_VEL
LIN {X 0,Y 326.602,Z 543.803,A -85,B 0,C 180,E1 -14907.455,E2 -14907.455} C_VEL
LIN {X 0,Y 326.655,Z 543.792,A -85,B 0,C 180,E1 -14910.34,E2 -14910.34} C_VEL
LIN {X 0,Y 326.684,Z 543.789,A -85,B 0,C 180,E1 -14914.516,E2 -14914.516} C_VEL
LIN {X 0,Y 326.613,Z 543.797,A -85,B 0,C 180,E1 -14918.543,E2 -14918.543} C_VEL
LIN {X 0,Y 326.738,Z 543.785,A -85,B 0,C 180,E1 -14921.177,E2 -14921.177} C_VEL
LIN {X 0,Y 326.756,Z 543.785,A -85,B 0,C 180,E1 -14925.433,E2 -14925.433} C_VEL
LIN {X 0,Y 326.762,Z 543.778,A -85,B 0,C 180,E1 -14928.839,E2 -14928.839} C_VEL
LIN {X 0,Y 326.96,Z 543.754,A -85,B 0,C 180,E1 -14932.59,E2 -14932.59} C_VEL
LIN {X 0,Y 326.771,Z 543.779,A -85,B 0,C 180,E1 -14935.065,E2 -14935.065} C_VEL
LIN {X 0,Y 327.04,Z 543.749,A -85,B 0,C 180,E1 -14937.537,E2 -14937.537} C_VEL
LIN {X 0,Y 327.19,Z 543.726,A -85,B 0,C 180,E1 -14940,E2 -14940} C_VEL
LIN {X 0,Y 327.041,Z 543.741,A -85,B 0,C 180,E1 -14942.463,E2 -14942.463} C_VEL
LIN {X 0,Y 326.953,Z 543.755,A -85,B 0,C 180,E1 -14946.639,E2 -14946.639} C_VEL
LIN {X 0,Y 326.798,Z 543.772,A -85,B 0,C 180,E1 -14949.907,E2 -14949.907} C_VEL
LIN {X 0,Y 326.752,Z 543.783,A -85,B 0,C 180,E1 -14953.686,E2 -14953.686} C_VEL
LIN {X 0,Y 326.692,Z 543.791,A -85,B 0,C 180,E1 -14957.529,E2 -14957.529} C_VEL
LIN {X 0,Y 326.656,Z 543.789,A -85,B 0,C 180,E1 -14960.136,E2 -14960.136} C_VEL
LIN {X 0,Y 326.646,Z 543.794,A -85,B 0,C 180,E1 -14964.13,E2 -14964.13} C_VEL
LIN {X 0,Y 326.68,Z 543.789,A -85,B 0,C 180,E1 -14966.858,E2 -14966.858} C_VEL
LIN {X 0,Y 326.634,Z 543.795,A -85,B 0,C 180,E1 -14970.612,E2 -14970.612} C_VEL
LIN {X 0,Y 326.603,Z 543.8,A -85,B 0,C 180,E1 -14974.02,E2 -14974.02} C_VEL
LIN {X 0,Y 326.625,Z 543.798,A -85,B 0,C 180,E1 -14977.24,E2 -14977.24} C_VEL
LIN {X 0,Y 326.576,Z 543.805,A -85,B 0,C 180,E1 -14981.132,E2 -14981.132} C_VEL
LIN {X 0,Y 326.584,Z 543.802,A -85,B 0,C 180,E1 -14984.754,E2 -14984.754} C_VEL
LIN {X 0,Y 326.62,Z 543.797,A -85,B 0,C 180,E1 -14988.162,E2 -14988.162} C_VEL
LIN {X 0,Y 326.646,Z 543.798,A -85,B 0,C 180,E1 -14991.396,E2 -14991.396} C_VEL
LIN {X 0,Y 326.619,Z 543.798,A -85,B 0,C 180,E1 -14994.852,E2 -14994.852} C_VEL
LIN {X 0,Y 326.608,Z 543.804,A -85,B 0,C 180,E1 -14997.456,E2 -14997.456} C_VEL
LIN {X 0,Y 326.661,Z 543.793,A -85,B 0,C 180,E1 -15000.342,E2 -15000.342} C_VEL
LIN {X 0,Y 326.691,Z 543.788,A -85,B 0,C 180,E1 -15004.517,E2 -15004.517} C_VEL
LIN {X 0,Y 326.672,Z 543.902,A -85,B 0,C 180,E1 -15007.133,E2 -15007.133} C_VEL
LIN {X 0,Y 328.626,Z 553.356,A -85,B 0,C 180,E1 -15010.16,E2 -15010.16} C_VEL
LIN {X 0,Y 333.56,Z 567.281,A -85,B 0,C 180,E1 -15010.826,E2 -15010.826} C_VEL
LIN {X 0,Y 336.364,Z 582.239,A -85,B 0,C 180,E1 -15011.353,E2 -15011.353} C_VEL
LIN {X 0,Y 334.852,Z 660.094,A -85,B 0,C 180,E1 -15013.031,E2 -15013.031} C_VEL
LIN {X 0,Y 334.286,Z 672.471,A -85,B 0,C 180,E1 -15013.512,E2 -15013.512} C_VEL
LIN {X 0,Y 333.437,Z 685.297,A -85,B 0,C 180,E1 -15014.254,E2 -15014.254} C_VEL
LIN {X 0,Y 332.407,Z 696.691,A -85,B 0,C 180,E1 -15015.146,E2 -15015.146} C_VEL
LIN {X 0,Y 331.282,Z 708.361,A -85,B 0,C 180,E1 -15016.349,E2 -15016.349} C_VEL
LIN {X 0,Y 330.015,Z 718.835,A -85,B 0,C 180,E1 -15017.704,E2 -15017.704} C_VEL
LIN {X 0,Y 328.757,Z 728.452,A -85,B 0,C 180,E1 -15019.251,E2 -15019.251} C_VEL
LIN {X 0,Y 327.745,Z 737.559,A -85,B 0,C 180,E1 -15021.104,E2 -15021.104} C_VEL
LIN {X 0,Y 326.761,Z 744.671,A -85,B 0,C 180,E1 -15022.896,E2 -15022.896} C_VEL
LIN {X 0,Y 325.923,Z 751.402,A -85,B 0,C 180,E1 -15025.052,E2 -15025.052} C_VEL
LIN {X 0,Y 325.53,Z 755.84,A -85,B 0,C 180,E1 -15026.906,E2 -15026.906} C_VEL
LIN {X 0,Y 325.081,Z 759.226,A -85,B 0,C 180,E1 -15028.761,E2 -15028.761} C_VEL
LIN {X 0,Y 324.952,Z 760.906,A -85,B 0,C 180,E1 -15030,E2 -15030} C_VEL
LIN {X 0,Y 324.866,Z 763.082,A -85,B 0,C 180,E1 -15032.48,E2 -15032.48} C_VEL
LIN {X 0,Y 324.922,Z 763.565,A -85,B 0,C 180,E1 -15033.72,E2 -15033.72} C_VEL
LIN {X 0,Y 324.949,Z 763.333,A -85,B 0,C 180,E1 -15036.208,E2 -15036.208} C_VEL
LIN {X 0,Y 324.977,Z 762.646,A -85,B 0,C 180,E1 -15037.455,E2 -15037.455} C_VEL
LIN {X 0,Y 325.107,Z 761.545,A -85,B 0,C 180,E1 -15038.703,E2 -15038.703} C_VEL
LIN {X 0,Y 325.281,Z 760.005,A -85,B 0,C 180,E1 -15039.953,E2 -15039.953} C_VEL
LIN {X 0,Y 325.739,Z 756.904,A -85,B 0,C 180,E1 -15041.827,E2 -15041.827} C_VEL
LIN {X 0,Y 326.351,Z 752.737,A -85,B 0,C 180,E1 -15043.702,E2 -15043.702} C_VEL
LIN {X 0,Y 327.343,Z 746.37,A -85,B 0,C 180,E1 -15045.887,E2 -15045.887} C_VEL
LIN {X 0,Y 328.527,Z 739.405,A -85,B 0,C 180,E1 -15047.748,E2 -15047.748} C_VEL
LIN {X 0,Y 330.046,Z 730.646,A -85,B 0,C 180,E1 -15049.595,E2 -15049.595} C_VEL
LIN {X 0,Y 331.336,Z 721.653,A -85,B 0,C 180,E1 -15051.136,E2 -15051.136} C_VEL
LIN {X 0,Y 332.727,Z 711.737,A -85,B 0,C 180,E1 -15052.509,E2 -15052.509} C_VEL
LIN {X 0,Y 334.142,Z 700.706,A -85,B 0,C 180,E1 -15053.719,E2 -15053.719} C_VEL
LIN {X 0,Y 335.502,Z 688.315,A -85,B 0,C 180,E1 -15054.768,E2 -15054.768} C_VEL
LIN {X 0,Y 336.416,Z 676.513,A -85,B 0,C 180,E1 -15055.522,E2 -15055.522} C_VEL
LIN {X 0,Y 337.232,Z 663.654,A -85,B 0,C 180,E1 -15056.079,E2 -15056.079} C_VEL
LIN {X 0,Y 337.79,Z 645.182,A -85,B 0,C 180,E1 -15056.536,E2 -15056.536} C_VEL
LIN {X 0,Y 339.149,Z 583.783,A -85,B 0,C 180,E1 -15057.837,E2 -15057.837} C_VEL
LIN {X 0,Y 336.498,Z 571.945,A -85,B 0,C 180,E1 -15058.33,E2 -15058.33} C_VEL
LIN {X 0,Y 329.907,Z 556.204,A -85,B 0,C 180,E1 -15059.27,E2 -15059.27} C_VEL
LIN {X 0,Y 328.704,Z 553.338,A -85,B 0,C 180,E1 -15059.456,E2 -15059.456} C_VEL
LIN {X 0,Y 327.572,Z 547.95,A -85,B 0,C 180,E1 -15061.298,E2 -15061.298} C_VEL
LIN {X 0,Y 326.523,Z 546.462,A -85,B 0,C 180,E1 -15061.923,E2 -15061.923} C_VEL
LIN {X 0,Y 323.265,Z 545.129,A -85,B 0,C 180,E1 -15062.946,E2 -15062.946} C_VEL
LIN {X 0,Y 320.23,Z 544.715,A -85,B 0,C 180,E1 -15064.029,E2 -15064.029} C_VEL
LIN {X 0,Y 319.551,Z 544.679,A -85,B 0,C 180,E1 -15064.739,E2 -15064.739} C_VEL
LIN {X 0,Y 319.583,Z 544.672,A -85,B 0,C 180,E1 -15068.005,E2 -15068.005} C_VEL
LIN {X 0,Y 319.595,Z 544.673,A -85,B 0,C 180,E1 -15071.61,E2 -15071.61} C_VEL
LIN {X 0,Y 319.577,Z 544.675,A -85,B 0,C 180,E1 -15075.272,E2 -15075.272} C_VEL
LIN {X 0,Y 319.543,Z 544.668,A -85,B 0,C 180,E1 -15078.714,E2 -15078.714} C_VEL
LIN {X 0,Y 319.595,Z 544.675,A -85,B 0,C 180,E1 -15082.338,E2 -15082.338} C_VEL
LIN {X 0,Y 319.556,Z 544.678,A -85,B 0,C 180,E1 -15085.123,E2 -15085.123} C_VEL
LIN {X 0,Y 319.566,Z 544.673,A -85,B 0,C 180,E1 -15089.057,E2 -15089.057} C_VEL
LIN {X 0,Y 319.604,Z 544.672,A -85,B 0,C 180,E1 -15092.497,E2 -15092.497} C_VEL
LIN {X 0,Y 319.599,Z 544.673,A -85,B 0,C 180,E1 -15095.303,E2 -15095.303} C_VEL
LIN {X 0,Y 319.592,Z 544.666,A -85,B 0,C 180,E1 -15098.047,E2 -15098.047} C_VEL
LIN {X 0,Y 319.683,Z 544.66,A -85,B 0,C 180,E1 -15100.962,E2 -15100.962} C_VEL
LIN {X 0,Y 319.724,Z 544.657,A -85,B 0,C 180,E1 -15105.276,E2 -15105.276} C_VEL
LIN {X 0,Y 319.745,Z 544.655,A -85,B 0,C 180,E1 -15109.872,E2 -15109.872} C_VEL
LIN {X 0,Y 319.906,Z 544.628,A -85,B 0,C 180,E1 -15112.425,E2 -15112.425} C_VEL
LIN {X 0,Y 319.74,Z 544.657,A -85,B 0,C 180,E1 -15114.956,E2 -15114.956} C_VEL
LIN {X 0,Y 319.985,Z 544.615,A -85,B 0,C 180,E1 -15117.482,E2 -15117.482} C_VEL
LIN {X 0,Y 320.162,Z 544.602,A -85,B 0,C 180,E1 -15120,E2 -15120} C_VEL
LIN {X 0,Y 319.984,Z 544.619,A -85,B 0,C 180,E1 -15122.518,E2 -15122.518} C_VEL
LIN {X 0,Y 319.936,Z 544.633,A -85,B 0,C 180,E1 -15126.306,E2 -15126.306} C_VEL
LIN {X 0,Y 319.83,Z 544.638,A -85,B 0,C 180,E1 -15128.848,E2 -15128.848} C_VEL
LIN {X 0,Y 319.674,Z 544.658,A -85,B 0,C 180,E1 -15132.7,E2 -15132.7} C_VEL
LIN {X 0,Y 319.692,Z 544.661,A -85,B 0,C 180,E1 -15135.296,E2 -15135.296} C_VEL
LIN {X 0,Y 319.667,Z 544.663,A -85,B 0,C 180,E1 -15139.255,E2 -15139.255} C_VEL
LIN {X 0,Y 319.554,Z 544.674,A -85,B 0,C 180,E1 -15143.321,E2 -15143.321} C_VEL
LIN {X 0,Y 319.629,Z 544.67,A -85,B 0,C 180,E1 -15146.089,E2 -15146.089} C_VEL
LIN {X 0,Y 319.584,Z 544.676,A -85,B 0,C 180,E1 -15148.934,E2 -15148.934} C_VEL
LIN {X 0,Y 319.527,Z 544.682,A -85,B 0,C 180,E1 -15151.862,E2 -15151.862} C_VEL
LIN {X 0,Y 319.575,Z 544.676,A -85,B 0,C 180,E1 -15155.544,E2 -15155.544} C_VEL
LIN {X 0,Y 319.578,Z 544.676,A -85,B 0,C 180,E1 -15158.007,E2 -15158.007} C_VEL
LIN {X 0,Y 319.568,Z 544.678,A -85,B 0,C 180,E1 -15161.607,E2 -15161.607} C_VEL
LIN {X 0,Y 319.519,Z 544.684,A -85,B 0,C 180,E1 -15165.264,E2 -15165.264} C_VEL
LIN {X 0,Y 319.526,Z 544.686,A -85,B 0,C 180,E1 -15168.713,E2 -15168.713} C_VEL
LIN {X 0,Y 319.559,Z 544.677,A -85,B 0,C 180,E1 -15172.349,E2 -15172.349} C_VEL
LIN {X 0,Y 319.567,Z 544.677,A -85,B 0,C 180,E1 -15175.89,E2 -15175.89} C_VEL
LIN {X 0,Y 319.582,Z 544.908,A -85,B 0,C 180,E1 -15176.479,E2 -15176.479} C_VEL
LIN {X 0,Y 322.077,Z 555.273,A -85,B 0,C 180,E1 -15179.876,E2 -15179.876} C_VEL
LIN {X 0,Y 324.333,Z 566.312,A -85,B 0,C 180,E1 -15183.281,E2 -15183.281} C_VEL
LIN {X 0,Y 324.799,Z 569.631,A -85,B 0,C 180,E1 -15184.24,E2 -15184.24} C_VEL
LIN {X 0,Y 329.282,Z 591.756,A -85,B 0,C 180,E1 -15185.17,E2 -15185.17} C_VEL
LIN {X 0,Y 332.203,Z 609.273,A -85,B 0,C 180,E1 -15185.831,E2 -15185.831} C_VEL
LIN {X 0,Y 330.557,Z 678.005,A -85,B 0,C 180,E1 -15187.343,E2 -15187.343} C_VEL
LIN {X 0,Y 329.676,Z 691.75,A -85,B 0,C 180,E1 -15187.89,E2 -15187.89} C_VEL
LIN {X 0,Y 328.414,Z 704.763,A -85,B 0,C 180,E1 -15188.667,E2 -15188.667} C_VEL
LIN {X 0,Y 327.025,Z 717.338,A -85,B 0,C 180,E1 -15189.725,E2 -15189.725} C_VEL
LIN {X 0,Y 325.399,Z 728.551,A -85,B 0,C 180,E1 -15190.934,E2 -15190.934} C_VEL
LIN {X 0,Y 323.835,Z 738.66,A -85,B 0,C 180,E1 -15192.312,E2 -15192.312} C_VEL
LIN {X 0,Y 322.419,Z 747.782,A -85,B 0,C 180,E1 -15193.864,E2 -15193.864} C_VEL
LIN {X 0,Y 321.007,Z 756.684,A -85,B 0,C 180,E1 -15195.742,E2 -15195.742} C_VEL
LIN {X 0,Y 319.753,Z 763.857,A -85,B 0,C 180,E1 -15197.626,E2 -15197.626} C_VEL
LIN {X 0,Y 319.05,Z 768.707,A -85,B 0,C 180,E1 -15199.209,E2 -15199.209} C_VEL
LIN {X 0,Y 318.411,Z 773.43,A -85,B 0,C 180,E1 -15201.112,E2 -15201.112} C_VEL
LIN {X 0,Y 317.996,Z 777.047,A -85,B 0,C 180,E1 -15203.018,E2 -15203.018} C_VEL
LIN {X 0,Y 317.806,Z 779.663,A -85,B 0,C 180,E1 -15204.925,E2 -15204.925} C_VEL
LIN {X 0,Y 317.807,Z 780.903,A -85,B 0,C 180,E1 -15206.196,E2 -15206.196} C_VEL
LIN {X 0,Y 317.758,Z 781.719,A -85,B 0,C 180,E1 -15207.465,E2 -15207.465} C_VEL
LIN {X 0,Y 317.782,Z 782.133,A -85,B 0,C 180,E1 -15210,E2 -15210} C_VEL
LIN {X 0,Y 317.745,Z 781.76,A -85,B 0,C 180,E1 -15211.267,E2 -15211.267} C_VEL
LIN {X 0,Y 317.76,Z 780.981,A -85,B 0,C 180,E1 -15212.535,E2 -15212.535} C_VEL
LIN {X 0,Y 317.808,Z 779.765,A -85,B 0,C 180,E1 -15213.804,E2 -15213.804} C_VEL
LIN {X 0,Y 317.839,Z 777.17,A -85,B 0,C 180,E1 -15215.712,E2 -15215.712} C_VEL
LIN {X 0,Y 318.072,Z 773.561,A -85,B 0,C 180,E1 -15217.618,E2 -15217.618} C_VEL
LIN {X 0,Y 318.496,Z 768.833,A -85,B 0,C 180,E1 -15219.526,E2 -15219.526} C_VEL
LIN {X 0,Y 319.264,Z 761.718,A -85,B 0,C 180,E1 -15221.749,E2 -15221.749} C_VEL
LIN {X 0,Y 320.339,Z 753.998,A -85,B 0,C 180,E1 -15223.641,E2 -15223.641} C_VEL
LIN {X 0,Y 321.57,Z 744.776,A -85,B 0,C 180,E1 -15225.441,E2 -15225.441} C_VEL
LIN {X 0,Y 322.662,Z 735.338,A -85,B 0,C 180,E1 -15226.937,E2 -15226.937} C_VEL
LIN {X 0,Y 323.989,Z 724.351,A -85,B 0,C 180,E1 -15228.332,E2 -15228.332} C_VEL
LIN {X 0,Y 325.175,Z 713.573,A -85,B 0,C 180,E1 -15229.408,E2 -15229.408} C_VEL
LIN {X 0,Y 326.269,Z 701.711,A -85,B 0,C 180,E1 -15230.324,E2 -15230.324} C_VEL
LIN {X 0,Y 327.246,Z 688.949,A -85,B 0,C 180,E1 -15231.042,E2 -15231.042} C_VEL
LIN {X 0,Y 327.927,Z 676.197,A -85,B 0,C 180,E1 -15231.503,E2 -15231.503} C_VEL
LIN {X 0,Y 329.24,Z 608.08,A -85,B 0,C 180,E1 -15232.993,E2 -15232.993} C_VEL
LIN {X 0,Y 324.193,Z 575.028,A -85,B 0,C 180,E1 -15234.111,E2 -15234.111} C_VEL
LIN {X 0,Y 323.295,Z 569.65,A -85,B 0,C 180,E1 -15234.328,E2 -15234.328} C_VEL
LIN {X 0,Y 323.706,Z 565.654,A -85,B 0,C 180,E1 -15235.39,E2 -15235.39} C_VEL
LIN {X 0,Y 321.94,Z 555.462,A -85,B 0,C 180,E1 -15238.346,E2 -15238.346} C_VEL
LIN {X 0,Y 319.579,Z 544.68,A -85,B 0,C 180,E1 -15241.674,E2 -15241.674} C_VEL
LIN {X 0,Y 319.579,Z 544.677,A -85,B 0,C 180,E1 -15245.542,E2 -15245.542} C_VEL
LIN {X 0,Y 319.572,Z 544.677,A -85,B 0,C 180,E1 -15248.007,E2 -15248.007} C_VEL
LIN {X 0,Y 319.523,Z 544.685,A -85,B 0,C 180,E1 -15251.596,E2 -15251.596} C_VEL
LIN {X 0,Y 319.548,Z 544.681,A -85,B 0,C 180,E1 -15255.268,E2 -15255.268} C_VEL
LIN {X 0,Y 319.542,Z 544.679,A -85,B 0,C 180,E1 -15258.714,E2 -15258.714} C_VEL
LIN {X 0,Y 319.577,Z 544.674,A -85,B 0,C 180,E1 -15262.342,E2 -15262.342} C_VEL
LIN {X 0,Y 319.555,Z 544.679,A -85,B 0,C 180,E1 -15265.123,E2 -15265.123} C_VEL
LIN {X 0,Y 319.564,Z 544.677,A -85,B 0,C 180,E1 -15269.057,E2 -15269.057} C_VEL
LIN {X 0,Y 319.603,Z 544.669,A -85,B 0,C 180,E1 -15272.498,E2 -15272.498} C_VEL
LIN {X 0,Y 319.597,Z 544.676,A -85,B 0,C 180,E1 -15275.303,E2 -15275.303} C_VEL
LIN {X 0,Y 319.597,Z 544.677,A -85,B 0,C 180,E1 -15279.4,E2 -15279.4} C_VEL
LIN {X 0,Y 319.651,Z 544.663,A -85,B 0,C 180,E1 -15282.073,E2 -15282.073} C_VEL
LIN {X 0,Y 319.725,Z 544.657,A -85,B 0,C 180,E1 -15286.008,E2 -15286.008} C_VEL
LIN {X 0,Y 319.749,Z 544.654,A -85,B 0,C 180,E1 -15289.873,E2 -15289.873} C_VEL
LIN {X 0,Y 319.919,Z 544.631,A -85,B 0,C 180,E1 -15292.426,E2 -15292.426} C_VEL
LIN {X 0,Y 319.74,Z 544.654,A -85,B 0,C 180,E1 -15294.956,E2 -15294.956} C_VEL
LIN {X 0,Y 319.984,Z 544.628,A -85,B 0,C 180,E1 -15297.482,E2 -15297.482} C_VEL
LIN {X 0,Y 320.142,Z 544.604,A -85,B 0,C 180,E1 -15300,E2 -15300} C_VEL
LIN {X 0,Y 319.985,Z 544.62,A -85,B 0,C 180,E1 -15302.518,E2 -15302.518} C_VEL
LIN {X 0,Y 319.915,Z 544.631,A -85,B 0,C 180,E1 -15306.627,E2 -15306.627} C_VEL
LIN {X 0,Y 319.745,Z 544.648,A -85,B 0,C 180,E1 -15310.128,E2 -15310.128} C_VEL
LIN {X 0,Y 319.724,Z 544.656,A -85,B 0,C 180,E1 -15314.724,E2 -15314.724} C_VEL
LIN {X 0,Y 319.683,Z 544.661,A -85,B 0,C 180,E1 -15319.038,E2 -15319.038} C_VEL
LIN {X 0,Y 319.565,Z 544.68,A -85,B 0,C 180,E1 -15323.32,E2 -15323.32} C_VEL
LIN {X 0,Y 319.63,Z 544.667,A -85,B 0,C 180,E1 -15326.089,E2 -15326.089} C_VEL
LIN {X 0,Y 319.585,Z 544.675,A -85,B 0,C 180,E1 -15328.934,E2 -15328.934} C_VEL
LIN {X 0,Y 319.528,Z 544.682,A -85,B 0,C 180,E1 -15331.863,E2 -15331.863} C_VEL
LIN {X 0,Y 319.577,Z 544.676,A -85,B 0,C 180,E1 -15335.544,E2 -15335.544} C_VEL
LIN {X 0,Y 319.555,Z 544.674,A -85,B 0,C 180,E1 -15338.011,E2 -15338.011} C_VEL
LIN {X 0,Y 319.549,Z 544.681,A -85,B 0,C 180,E1 -15341.603,E2 -15341.603} C_VEL
LIN {X 0,Y 319.575,Z 544.679,A -85,B 0,C 180,E1 -15345.274,E2 -15345.274} C_VEL
LIN {X 0,Y 319.577,Z 544.674,A -85,B 0,C 180,E1 -15348.721,E2 -15348.721} C_VEL
LIN {X 0,Y 319.598,Z 544.672,A -85,B 0,C 180,E1 -15352.34,E2 -15352.34} C_VEL
LIN {X 0,Y 319.56,Z 544.68,A -85,B 0,C 180,E1 -15355.124,E2 -15355.124} C_VEL
LIN {X 0,Y 319.57,Z 544.679,A -85,B 0,C 180,E1 -15359.059,E2 -15359.059} C_VEL
LIN {X 0,Y 319.609,Z 544.672,A -85,B 0,C 180,E1 -15362.499,E2 -15362.499} C_VEL
LIN {X 0,Y 319.607,Z 544.675,A -85,B 0,C 180,E1 -15365.305,E2 -15365.305} C_VEL
LIN {X 0,Y 319.647,Z 544.875,A -85,B 0,C 180,E1 -15366.789,E2 -15366.789} C_VEL
LIN {X 0,Y 321.41,Z 553.381,A -85,B 0,C 180,E1 -15369.629,E2 -15369.629} C_VEL
LIN {X 0,Y 327.155,Z 569.349,A -85,B 0,C 180,E1 -15370.426,E2 -15370.426} C_VEL
LIN {X 0,Y 329.734,Z 583.096,A -85,B 0,C 180,E1 -15370.924,E2 -15370.924} C_VEL
LIN {X 0,Y 328.14,Z 660.688,A -85,B 0,C 180,E1 -15372.632,E2 -15372.632} C_VEL
LIN {X 0,Y 327.536,Z 673.689,A -85,B 0,C 180,E1 -15373.162,E2 -15373.162} C_VEL
LIN {X 0,Y 326.643,Z 686.256,A -85,B 0,C 180,E1 -15373.918,E2 -15373.918} C_VEL
LIN {X 0,Y 325.6,Z 697.444,A -85,B 0,C 180,E1 -15374.829,E2 -15374.829} C_VEL
LIN {X 0,Y 324.413,Z 708.997,A -85,B 0,C 180,E1 -15376.054,E2 -15376.054} C_VEL
LIN {X 0,Y 323.123,Z 719.396,A -85,B 0,C 180,E1 -15377.438,E2 -15377.438} C_VEL
LIN {X 0,Y 321.816,Z 728.937,A -85,B 0,C 180,E1 -15379.016,E2 -15379.016} C_VEL
LIN {X 0,Y 320.848,Z 737.428,A -85,B 0,C 180,E1 -15380.779,E2 -15380.779} C_VEL
LIN {X 0,Y 319.74,Z 745.062,A -85,B 0,C 180,E1 -15382.739,E2 -15382.739} C_VEL
LIN {X 0,Y 319.167,Z 749.995,A -85,B 0,C 180,E1 -15384.313,E2 -15384.313} C_VEL
LIN {X 0,Y 318.807,Z 753.336,A -85,B 0,C 180,E1 -15385.575,E2 -15385.575} C_VEL
LIN {X 0,Y 318.157,Z 757.39,A -85,B 0,C 180,E1 -15387.468,E2 -15387.468} C_VEL
LIN {X 0,Y 317.988,Z 759.506,A -85,B 0,C 180,E1 -15388.734,E2 -15388.734} C_VEL
LIN {X 0,Y 317.79,Z 762.44,A -85,B 0,C 180,E1 -15391.267,E2 -15391.267} C_VEL
LIN {X 0,Y 317.786,Z 763.32,A -85,B 0,C 180,E1 -15392.535,E2 -15392.535} C_VEL
LIN {X 0,Y 317.827,Z 763.777,A -85,B 0,C 180,E1 -15393.804,E2 -15393.804} C_VEL
LIN {X 0,Y 317.873,Z 763.518,A -85,B 0,C 180,E1 -15396.347,E2 -15396.347} C_VEL
LIN {X 0,Y 317.914,Z 762.817,A -85,B 0,C 180,E1 -15397.622,E2 -15397.622} C_VEL
LIN {X 0,Y 318.046,Z 761.689,A -85,B 0,C 180,E1 -15398.898,E2 -15398.898} C_VEL
LIN {X 0,Y 318.249,Z 760.134,A -85,B 0,C 180,E1 -15400.175,E2 -15400.175} C_VEL
LIN {X 0,Y 318.743,Z 757.005,A -85,B 0,C 180,E1 -15402.091,E2 -15402.091} C_VEL
LIN {X 0,Y 319.409,Z 752.806,A -85,B 0,C 180,E1 -15404.006,E2 -15404.006} C_VEL
LIN {X 0,Y 320.465,Z 746.406,A -85,B 0,C 180,E1 -15406.237,E2 -15406.237} C_VEL
LIN {X 0,Y 321.711,Z 739.386,A -85,B 0,C 180,E1 -15408.137,E2 -15408.137} C_VEL
LIN {X 0,Y 323.309,Z 730.577,A -85,B 0,C 180,E1 -15410.021,E2 -15410.021} C_VEL
LIN {X 0,Y 324.667,Z 721.53,A -85,B 0,C 180,E1 -15411.591,E2 -15411.591} C_VEL
LIN {X 0,Y 326.138,Z 711.532,A -85,B 0,C 180,E1 -15412.99,E2 -15412.99} C_VEL
LIN {X 0,Y 327.613,Z 700.379,A -85,B 0,C 180,E1 -15414.221,E2 -15414.221} C_VEL
LIN {X 0,Y 329.024,Z 687.85,A -85,B 0,C 180,E1 -15415.29,E2 -15415.29} C_VEL
LIN {X 0,Y 329.875,Z 677.151,A -85,B 0,C 180,E1 -15415.981,E2 -15415.981} C_VEL
LIN {X 0,Y 330.744,Z 664.73,A -85,B 0,C 180,E1 -15416.542,E2 -15416.542} C_VEL
LIN {X 0,Y 331.281,Z 648.852,A -85,B 0,C 180,E1 -15416.961,E2 -15416.961} C_VEL
LIN {X 0,Y 332.76,Z 584.879,A -85,B 0,C 180,E1 -15418.341,E2 -15418.341} C_VEL
LIN {X 0,Y 330.33,Z 574.315,A -85,B 0,C 180,E1 -15418.8,E2 -15418.8} C_VEL
LIN {X 0,Y 324.114,Z 559.493,A -85,B 0,C 180,E1 -15419.716,E2 -15419.716} C_VEL
LIN {X 0,Y 321.533,Z 553.564,A -85,B 0,C 180,E1 -15420.11,E2 -15420.11} C_VEL
LIN {X 0,Y 319.566,Z 544.678,A -85,B 0,C 180,E1 -15423.353,E2 -15423.353} C_VEL
LIN {X 0,Y 319.551,Z 544.679,A -85,B 0,C 180,E1 -15424.739,E2 -15424.739} C_VEL
LIN {X 0,Y 318.933,Z 544.761,A -85,B 0,C 180,E1 -15425.791,E2 -15425.791} C_VEL
LIN {X 0,Y 316.099,Z 545.115,A -85,B 0,C 180,E1 -15427.504,E2 -15427.504} C_VEL
LIN {X 0,Y 313.664,Z 545.415,A -85,B 0,C 180,E1 -15428.893,E2 -15428.893} C_VEL
LIN {X 0,Y 312.611,Z 545.545,A -85,B 0,C 180,E1 -15429.968,E2 -15429.968} C_VEL
LIN {X 0,Y 312.524,Z 545.556,A -85,B 0,C 180,E1 -15430.332,E2 -15430.332} C_VEL
LIN {X 0,Y 312.534,Z 545.554,A -85,B 0,C 180,E1 -15434.193,E2 -15434.193} C_VEL
LIN {X 0,Y 312.53,Z 545.548,A -85,B 0,C 180,E1 -15437.908,E2 -15437.908} C_VEL
LIN {X 0,Y 312.554,Z 545.551,A -85,B 0,C 180,E1 -15441.904,E2 -15441.904} C_VEL
LIN {X 0,Y 312.502,Z 545.555,A -85,B 0,C 180,E1 -15445.789,E2 -15445.789} C_VEL
LIN {X 0,Y 312.519,Z 545.552,A -85,B 0,C 180,E1 -15448.853,E2 -15448.853} C_VEL
LIN {X 0,Y 312.57,Z 545.549,A -85,B 0,C 180,E1 -15451.824,E2 -15451.824} C_VEL
LIN {X 0,Y 312.58,Z 545.547,A -85,B 0,C 180,E1 -15454.71,E2 -15454.71} C_VEL
LIN {X 0,Y 312.582,Z 545.539,A -85,B 0,C 180,E1 -15457.528,E2 -15457.528} C_VEL
LIN {X 0,Y 312.632,Z 545.536,A -85,B 0,C 180,E1 -15461.656,E2 -15461.656} C_VEL
LIN {X 0,Y 312.687,Z 545.532,A -85,B 0,C 180,E1 -15465.686,E2 -15465.686} C_VEL
LIN {X 0,Y 312.691,Z 545.533,A -85,B 0,C 180,E1 -15469.641,E2 -15469.641} C_VEL
LIN {X 0,Y 312.846,Z 545.507,A -85,B 0,C 180,E1 -15472.253,E2 -15472.253} C_VEL
LIN {X 0,Y 312.71,Z 545.534,A -85,B 0,C 180,E1 -15474.842,E2 -15474.842} C_VEL
LIN {X 0,Y 312.985,Z 545.491,A -85,B 0,C 180,E1 -15478.713,E2 -15478.713} C_VEL
LIN {X 0,Y 313.114,Z 545.48,A -85,B 0,C 180,E1 -15480,E2 -15480} C_VEL
LIN {X 0,Y 312.93,Z 545.497,A -85,B 0,C 180,E1 -15482.574,E2 -15482.574} C_VEL
LIN {X 0,Y 312.893,Z 545.511,A -85,B 0,C 180,E1 -15486.448,E2 -15486.448} C_VEL
LIN {X 0,Y 312.76,Z 545.519,A -85,B 0,C 180,E1 -15489.05,E2 -15489.05} C_VEL
LIN {X 0,Y 312.627,Z 545.533,A -85,B 0,C 180,E1 -15492.991,E2 -15492.991} C_VEL
LIN {X 0,Y 312.631,Z 545.54,A -85,B 0,C 180,E1 -15495.65,E2 -15495.65} C_VEL
LIN {X 0,Y 312.623,Z 545.54,A -85,B 0,C 180,E1 -15499.236,E2 -15499.236} C_VEL
LIN {X 0,Y 312.519,Z 545.549,A -85,B 0,C 180,E1 -15502.781,E2 -15502.781} C_VEL
LIN {X 0,Y 312.597,Z 545.545,A -85,B 0,C 180,E1 -15505.936,E2 -15505.936} C_VEL
LIN {X 0,Y 312.54,Z 545.552,A -85,B 0,C 180,E1 -15509.65,E2 -15509.65} C_VEL
LIN {X 0,Y 312.514,Z 545.555,A -85,B 0,C 180,E1 -15513.689,E2 -15513.689} C_VEL
LIN {X 0,Y 312.536,Z 545.553,A -85,B 0,C 180,E1 -15517.384,E2 -15517.384} C_VEL
LIN {X 0,Y 312.498,Z 545.561,A -85,B 0,C 180,E1 -15520.708,E2 -15520.708} C_VEL
LIN {X 0,Y 312.515,Z 545.559,A -85,B 0,C 180,E1 -15524.198,E2 -15524.198} C_VEL
LIN {X 0,Y 312.483,Z 545.562,A -85,B 0,C 180,E1 -15527.919,E2 -15527.919} C_VEL
LIN {X 0,Y 312.503,Z 545.557,A -85,B 0,C 180,E1 -15531.918,E2 -15531.918} C_VEL
LIN {X 0,Y 312.538,Z 545.59,A -85,B 0,C 180,E1 -15535.847,E2 -15535.847} C_VEL
LIN {X 0,Y 315.308,Z 557.392,A -85,B 0,C 180,E1 -15539.815,E2 -15539.815} C_VEL
LIN {X 0,Y 317.404,Z 567.628,A -85,B 0,C 180,E1 -15543.05,E2 -15543.05} C_VEL
LIN {X 0,Y 317.778,Z 569.529,A -85,B 0,C 180,E1 -15543.583,E2 -15543.583} C_VEL
LIN {X 0,Y 319.471,Z 575.272,A -85,B 0,C 180,E1 -15543.886,E2 -15543.886} C_VEL
LIN {X 0,Y 324.423,Z 601.375,A -85,B 0,C 180,E1 -15544.978,E2 -15544.978} C_VEL
LIN {X 0,Y 325.842,Z 610.552,A -85,B 0,C 180,E1 -15545.323,E2 -15545.323} C_VEL
LIN {X 0,Y 324.098,Z 677.987,A -85,B 0,C 180,E1 -15546.832,E2 -15546.832} C_VEL
LIN {X 0,Y 323.185,Z 691.509,A -85,B 0,C 180,E1 -15547.38,E2 -15547.38} C_VEL
LIN {X 0,Y 321.942,Z 704.008,A -85,B 0,C 180,E1 -15548.132,E2 -15548.132} C_VEL
LIN {X 0,Y 320.584,Z 715.929,A -85,B 0,C 180,E1 -15549.131,E2 -15549.131} C_VEL
LIN {X 0,Y 318.861,Z 727.362,A -85,B 0,C 180,E1 -15550.36,E2 -15550.36} C_VEL
LIN {X 0,Y 317.238,Z 737.678,A -85,B 0,C 180,E1 -15551.765,E2 -15551.765} C_VEL
LIN {X 0,Y 315.863,Z 746.12,A -85,B 0,C 180,E1 -15553.187,E2 -15553.187} C_VEL
LIN {X 0,Y 314.368,Z 755.283,A -85,B 0,C 180,E1 -15555.103,E2 -15555.103} C_VEL
LIN {X 0,Y 312.975,Z 762.668,A -85,B 0,C 180,E1 -15557.024,E2 -15557.024} C_VEL
LIN {X 0,Y 312.051,Z 768.608,A -85,B 0,C 180,E1 -15558.964,E2 -15558.964} C_VEL
LIN {X 0,Y 311.384,Z 773.308,A -85,B 0,C 180,E1 -15560.91,E2 -15560.91} C_VEL
LIN {X 0,Y 310.929,Z 776.904,A -85,B 0,C 180,E1 -15562.859,E2 -15562.859} C_VEL
LIN {X 0,Y 310.71,Z 779.5,A -85,B 0,C 180,E1 -15564.809,E2 -15564.809} C_VEL
LIN {X 0,Y 310.718,Z 780.731,A -85,B 0,C 180,E1 -15566.109,E2 -15566.109} C_VEL
LIN {X 0,Y 310.681,Z 781.529,A -85,B 0,C 180,E1 -15567.407,E2 -15567.407} C_VEL
LIN {X 0,Y 310.692,Z 781.923,A -85,B 0,C 180,E1 -15570,E2 -15570} C_VEL
LIN {X 0,Y 310.659,Z 781.541,A -85,B 0,C 180,E1 -15571.296,E2 -15571.296} C_VEL
LIN {X 0,Y 310.683,Z 780.745,A -85,B 0,C 180,E1 -15572.593,E2 -15572.593} C_VEL
LIN {X 0,Y 310.719,Z 779.518,A -85,B 0,C 180,E1 -15573.891,E2 -15573.891} C_VEL
LIN {X 0,Y 310.748,Z 777.202,A -85,B 0,C 180,E1 -15575.661,E2 -15575.661} C_VEL
LIN {X 0,Y 311.014,Z 773.272,A -85,B 0,C 180,E1 -15577.792,E2 -15577.792} C_VEL
LIN {X 0,Y 311.448,Z 768.52,A -85,B 0,C 180,E1 -15579.744,E2 -15579.744} C_VEL
LIN {X 0,Y 312.288,Z 761.381,A -85,B 0,C 180,E1 -15582.015,E2 -15582.015} C_VEL
LIN {X 0,Y 313.415,Z 753.619,A -85,B 0,C 180,E1 -15583.949,E2 -15583.949} C_VEL
LIN {X 0,Y 314.672,Z 744.562,A -85,B 0,C 180,E1 -15585.751,E2 -15585.751} C_VEL
LIN {X 0,Y 315.844,Z 734.879,A -85,B 0,C 180,E1 -15587.314,E2 -15587.314} C_VEL
LIN {X 0,Y 317.195,Z 723.807,A -85,B 0,C 180,E1 -15588.739,E2 -15588.739} C_VEL
LIN {X 0,Y 318.466,Z 712.95,A -85,B 0,C 180,E1 -15589.834,E2 -15589.834} C_VEL
LIN {X 0,Y 319.613,Z 700.972,A -85,B 0,C 180,E1 -15590.767,E2 -15590.767} C_VEL
LIN {X 0,Y 320.646,Z 687.979,A -85,B 0,C 180,E1 -15591.496,E2 -15591.496} C_VEL
LIN {X 0,Y 321.296,Z 674.857,A -85,B 0,C 180,E1 -15591.962,E2 -15591.962} C_VEL
LIN {X 0,Y 322.599,Z 608.712,A -85,B 0,C 180,E1 -15593.434,E2 -15593.434} C_VEL
LIN {X 0,Y 317.679,Z 576.254,A -85,B 0,C 180,E1 -15594.562,E2 -15594.562} C_VEL
LIN {X 0,Y 316.495,Z 569.408,A -85,B 0,C 180,E1 -15594.851,E2 -15594.851} C_VEL
LIN {X 0,Y 316.737,Z 566.538,A -85,B 0,C 180,E1 -15595.637,E2 -15595.637} C_VEL
LIN {X 0,Y 314.925,Z 556.36,A -85,B 0,C 180,E1 -15598.672,E2 -15598.672} C_VEL
LIN {X 0,Y 312.537,Z 545.556,A -85,B 0,C 180,E1 -15602.086,E2 -15602.086} C_VEL
LIN {X 0,Y 312.534,Z 545.554,A -85,B 0,C 180,E1 -15605.949,E2 -15605.949} C_VEL
LIN {X 0,Y 312.506,Z 545.558,A -85,B 0,C 180,E1 -15609.027,E2 -15609.027} C_VEL
LIN {X 0,Y 312.49,Z 545.557,A -85,B 0,C 180,E1 -15612.43,E2 -15612.43} C_VEL
LIN {X 0,Y 312.52,Z 545.554,A -85,B 0,C 180,E1 -15616.022,E2 -15616.022} C_VEL
LIN {X 0,Y 312.507,Z 545.557,A -85,B 0,C 180,E1 -15619.872,E2 -15619.872} C_VEL
LIN {X 0,Y 312.536,Z 545.551,A -85,B 0,C 180,E1 -15622.616,E2 -15622.616} C_VEL
LIN {X 0,Y 312.514,Z 545.553,A -85,B 0,C 180,E1 -15626.311,E2 -15626.311} C_VEL
LIN {X 0,Y 312.54,Z 545.55,A -85,B 0,C 180,E1 -15630.35,E2 -15630.35} C_VEL
LIN {X 0,Y 312.597,Z 545.545,A -85,B 0,C 180,E1 -15634.064,E2 -15634.064} C_VEL
LIN {X 0,Y 312.558,Z 545.552,A -85,B 0,C 180,E1 -15637.527,E2 -15637.527} C_VEL
LIN {X 0,Y 312.631,Z 545.54,A -85,B 0,C 180,E1 -15641.656,E2 -15641.656} C_VEL
LIN {X 0,Y 312.687,Z 545.536,A -85,B 0,C 180,E1 -15645.686,E2 -15645.686} C_VEL
LIN {X 0,Y 312.694,Z 545.535,A -85,B 0,C 180,E1 -15649.642,E2 -15649.642} C_VEL
LIN {X 0,Y 312.859,Z 545.511,A -85,B 0,C 180,E1 -15652.254,E2 -15652.254} C_VEL
LIN {X 0,Y 312.71,Z 545.529,A -85,B 0,C 180,E1 -15654.842,E2 -15654.842} C_VEL
LIN {X 0,Y 312.983,Z 545.496,A -85,B 0,C 180,E1 -15658.713,E2 -15658.713} C_VEL
LIN {X 0,Y 312.983,Z 545.499,A -85,B 0,C 180,E1 -15661.287,E2 -15661.287} C_VEL
LIN {X 0,Y 312.711,Z 545.532,A -85,B 0,C 180,E1 -15665.158,E2 -15665.158} C_VEL
LIN {X 0,Y 312.847,Z 545.514,A -85,B 0,C 180,E1 -15667.747,E2 -15667.747} C_VEL
LIN {X 0,Y 312.662,Z 545.536,A -85,B 0,C 180,E1 -15671.672,E2 -15671.672} C_VEL
LIN {X 0,Y 312.694,Z 545.533,A -85,B 0,C 180,E1 -15674.888,E2 -15674.888} C_VEL
LIN {X 0,Y 312.624,Z 545.54,A -85,B 0,C 180,E1 -15679.237,E2 -15679.237} C_VEL
LIN {X 0,Y 312.54,Z 545.55,A -85,B 0,C 180,E1 -15682.79,E2 -15682.79} C_VEL
LIN {X 0,Y 312.598,Z 545.543,A -85,B 0,C 180,E1 -15685.936,E2 -15685.936} C_VEL
LIN {X 0,Y 312.541,Z 545.554,A -85,B 0,C 180,E1 -15689.651,E2 -15689.651} C_VEL
LIN {X 0,Y 312.515,Z 545.557,A -85,B 0,C 180,E1 -15693.69,E2 -15693.69} C_VEL
LIN {X 0,Y 312.534,Z 545.55,A -85,B 0,C 180,E1 -15697.384,E2 -15697.384} C_VEL
LIN {X 0,Y 312.488,Z 545.558,A -85,B 0,C 180,E1 -15700.71,E2 -15700.71} C_VEL
LIN {X 0,Y 312.508,Z 545.555,A -85,B 0,C 180,E1 -15704.2,E2 -15704.2} C_VEL
LIN {X 0,Y 312.547,Z 545.551,A -85,B 0,C 180,E1 -15707.906,E2 -15707.906} C_VEL
LIN {X 0,Y 312.557,Z 545.55,A -85,B 0,C 180,E1 -15711.906,E2 -15711.906} C_VEL
LIN {X 0,Y 312.506,Z 545.558,A -85,B 0,C 180,E1 -15715.791,E2 -15715.791} C_VEL
LIN {X 0,Y 312.524,Z 545.555,A -85,B 0,C 180,E1 -15718.855,E2 -15718.855} C_VEL
LIN {X 0,Y 312.575,Z 545.55,A -85,B 0,C 180,E1 -15721.826,E2 -15721.826} C_VEL
LIN {X 0,Y 312.587,Z 545.546,A -85,B 0,C 180,E1 -15724.712,E2 -15724.712} C_VEL
LIN {X 0,Y 312.578,Z 545.573,A -85,B 0,C 180,E1 -15726.333,E2 -15726.333} C_VEL
LIN {X 0,Y 314.194,Z 553.546,A -85,B 0,C 180,E1 -15729.073,E2 -15729.073} C_VEL
LIN {X 0,Y 320.781,Z 571.41,A -85,B 0,C 180,E1 -15730.011,E2 -15730.011} C_VEL
LIN {X 0,Y 323.123,Z 584.261,A -85,B 0,C 180,E1 -15730.486,E2 -15730.486} C_VEL
LIN {X 0,Y 321.504,Z 660.134,A -85,B 0,C 180,E1 -15732.18,E2 -15732.18} C_VEL
LIN {X 0,Y 320.9,Z 673.385,A -85,B 0,C 180,E1 -15732.721,E2 -15732.721} C_VEL
LIN {X 0,Y 319.956,Z 686.086,A -85,B 0,C 180,E1 -15733.491,E2 -15733.491} C_VEL
LIN {X 0,Y 318.799,Z 698.173,A -85,B 0,C 180,E1 -15734.497,E2 -15734.497} C_VEL
LIN {X 0,Y 317.554,Z 709.631,A -85,B 0,C 180,E1 -15735.747,E2 -15735.747} C_VEL
LIN {X 0,Y 316.242,Z 719.955,A -85,B 0,C 180,E1 -15737.16,E2 -15737.16} C_VEL
LIN {X 0,Y 314.877,Z 729.413,A -85,B 0,C 180,E1 -15738.771,E2 -15738.771} C_VEL
LIN {X 0,Y 313.854,Z 738.051,A -85,B 0,C 180,E1 -15740.618,E2 -15740.618} C_VEL
LIN {X 0,Y 312.725,Z 745.452,A -85,B 0,C 180,E1 -15742.576,E2 -15742.576} C_VEL
LIN {X 0,Y 312.113,Z 750.35,A -85,B 0,C 180,E1 -15744.184,E2 -15744.184} C_VEL
LIN {X 0,Y 311.746,Z 753.675,A -85,B 0,C 180,E1 -15745.475,E2 -15745.475} C_VEL
LIN {X 0,Y 311.073,Z 757.698,A -85,B 0,C 180,E1 -15747.41,E2 -15747.41} C_VEL
LIN {X 0,Y 310.895,Z 759.785,A -85,B 0,C 180,E1 -15748.705,E2 -15748.705} C_VEL
LIN {X 0,Y 310.702,Z 762.691,A -85,B 0,C 180,E1 -15751.296,E2 -15751.296} C_VEL
LIN {X 0,Y 310.708,Z 763.554,A -85,B 0,C 180,E1 -15752.593,E2 -15752.593} C_VEL
LIN {X 0,Y 310.735,Z 763.988,A -85,B 0,C 180,E1 -15753.891,E2 -15753.891} C_VEL
LIN {X 0,Y 310.799,Z 763.702,A -85,B 0,C 180,E1 -15756.492,E2 -15756.492} C_VEL
LIN {X 0,Y 310.846,Z 762.987,A -85,B 0,C 180,E1 -15757.796,E2 -15757.796} C_VEL
LIN {X 0,Y 311.002,Z 761.833,A -85,B 0,C 180,E1 -15759.101,E2 -15759.101} C_VEL
LIN {X 0,Y 311.209,Z 760.265,A -85,B 0,C 180,E1 -15760.408,E2 -15760.408} C_VEL
LIN {X 0,Y 311.758,Z 757.106,A -85,B 0,C 180,E1 -15762.366,E2 -15762.366} C_VEL
LIN {X 0,Y 312.469,Z 752.876,A -85,B 0,C 180,E1 -15764.324,E2 -15764.324} C_VEL
LIN {X 0,Y 313.585,Z 746.442,A -85,B 0,C 180,E1 -15766.603,E2 -15766.603} C_VEL
LIN {X 0,Y 314.907,Z 739.364,A -85,B 0,C 180,E1 -15768.543,E2 -15768.543} C_VEL
LIN {X 0,Y 316.583,Z 730.51,A -85,B 0,C 180,E1 -15770.465,E2 -15770.465} C_VEL
LIN {X 0,Y 318.003,Z 721.408,A -85,B 0,C 180,E1 -15772.067,E2 -15772.067} C_VEL
